LIN {X 0,Y 573.388,Z 194.884,A -85,B 0,C 180,E1 -2263.851,E2 -2263.851} C_VEL
LIN {X 0,Y 573.533,Z 175.271,A -85,B 0,C 180,E1 -2266.721,E2 -2266.721} C_VEL
LIN {X 0,Y 573.704,Z 157.685,A -85,B 0,C 180,E1 -2269.315,E2 -2269.315} C_VEL
LIN {X 0,Y 573.895,Z 140.113,A -85,B 0,C 180,E1 -2271.932,E2 -2271.932} C_VEL
LIN {X 0,Y 573.247,Z 134.603,A -85,B 0,C 180,E1 -2272.789,E2 -2272.789} C_VEL
LIN {X 0,Y 573.229,Z 134.582,A -85,B 0,C 180,E1 -2275.411,E2 -2275.411} C_VEL
LIN {X 0,Y 573.202,Z 134.579,A -85,B 0,C 180,E1 -2278.019,E2 -2278.019} C_VEL
LIN {X 0,Y 573.22,Z 134.577,A -85,B 0,C 180,E1 -2280.178,E2 -2280.178} C_VEL
LIN {X 0,Y 573.246,Z 134.579,A -85,B 0,C 180,E1 -2282.645,E2 -2282.645} C_VEL
LIN {X 0,Y 573.203,Z 134.583,A -85,B 0,C 180,E1 -2285.188,E2 -2285.188} C_VEL
LIN {X 0,Y 573.23,Z 134.575,A -85,B 0,C 180,E1 -2287.808,E2 -2287.808} C_VEL
LIN {X 0,Y 573.245,Z 134.58,A -85,B 0,C 180,E1 -2290.525,E2 -2290.525} C_VEL
LIN {X 0,Y 573.208,Z 134.579,A -85,B 0,C 180,E1 -2293.362,E2 -2293.362} C_VEL
LIN {X 0,Y 573.235,Z 134.581,A -85,B 0,C 180,E1 -2296.332,E2 -2296.332} C_VEL
LIN {X 0,Y 573.245,Z 134.574,A -85,B 0,C 180,E1 -2299.475,E2 -2299.475} C_VEL
LIN {X 0,Y 573.229,Z 134.583,A -85,B 0,C 180,E1 -2302.192,E2 -2302.192} C_VEL
LIN {X 0,Y 573.232,Z 134.575,A -85,B 0,C 180,E1 -2305.229,E2 -2305.229} C_VEL
LIN {X 0,Y 573.246,Z 134.577,A -85,B 0,C 180,E1 -2307.772,E2 -2307.772} C_VEL
LIN {X 0,Y 573.242,Z 134.576,A -85,B 0,C 180,E1 -2310.633,E2 -2310.633} C_VEL
LIN {X 0,Y 573.208,Z 134.578,A -85,B 0,C 180,E1 -2313.022,E2 -2313.022} C_VEL
LIN {X 0,Y 573.274,Z 134.572,A -85,B 0,C 180,E1 -2315.366,E2 -2315.366} C_VEL
LIN {X 0,Y 573.227,Z 134.578,A -85,B 0,C 180,E1 -2318.419,E2 -2318.419} C_VEL
LIN {X 0,Y 573.268,Z 134.571,A -85,B 0,C 180,E1 -2320.731,E2 -2320.731} C_VEL
LIN {X 0,Y 573.242,Z 134.582,A -85,B 0,C 180,E1 -2323.621,E2 -2323.621} C_VEL
LIN {X 0,Y 573.272,Z 134.578,A -85,B 0,C 180,E1 -2325.807,E2 -2325.807} C_VEL
LIN {X 0,Y 573.263,Z 134.572,A -85,B 0,C 180,E1 -2328.745,E2 -2328.745} C_VEL
LIN {X 0,Y 573.283,Z 134.578,A -85,B 0,C 180,E1 -2331.54,E2 -2331.54} C_VEL
LIN {X 0,Y 573.291,Z 134.568,A -85,B 0,C 180,E1 -2334.372,E2 -2334.372} C_VEL
LIN {X 0,Y 573.316,Z 134.566,A -85,B 0,C 180,E1 -2337.892,E2 -2337.892} C_VEL
LIN {X 0,Y 573.325,Z 134.566,A -85,B 0,C 180,E1 -2340.702,E2 -2340.702} C_VEL
LIN {X 0,Y 573.299,Z 134.571,A -85,B 0,C 180,E1 -2342.811,E2 -2342.811} C_VEL
LIN {X 0,Y 573.298,Z 134.569,A -85,B 0,C 180,E1 -2345.628,E2 -2345.628} C_VEL
LIN {X 0,Y 573.282,Z 134.571,A -85,B 0,C 180,E1 -2348.46,E2 -2348.46} C_VEL
LIN {X 0,Y 573.272,Z 134.574,A -85,B 0,C 180,E1 -2351.312,E2 -2351.312} C_VEL
LIN {X 0,Y 573.282,Z 134.573,A -85,B 0,C 180,E1 -2354.424,E2 -2354.424} C_VEL
LIN {X 0,Y 573.258,Z 134.576,A -85,B 0,C 180,E1 -2357.112,E2 -2357.112} C_VEL
LIN {X 0,Y 573.252,Z 134.575,A -85,B 0,C 180,E1 -2360.077,E2 -2360.077} C_VEL
LIN {X 0,Y 573.235,Z 134.577,A -85,B 0,C 180,E1 -2363.1,E2 -2363.1} C_VEL
LIN {X 0,Y 573.249,Z 134.577,A -85,B 0,C 180,E1 -2364.376,E2 -2364.376} C_VEL
LIN {X 0,Y 572.622,Z 134.659,A -85,B 0,C 180,E1 -2364.962,E2 -2364.962} C_VEL
LIN {X 0,Y 569.782,Z 135.012,A -85,B 0,C 180,E1 -2365.914,E2 -2365.914} C_VEL
LIN {X 0,Y 567.351,Z 135.314,A -85,B 0,C 180,E1 -2366.679,E2 -2366.679} C_VEL
LIN {X 0,Y 566.295,Z 135.44,A -85,B 0,C 180,E1 -2367.27,E2 -2367.27} C_VEL
LIN {X 0,Y 566.204,Z 135.451,A -85,B 0,C 180,E1 -2367.471,E2 -2367.471} C_VEL
LIN {X 0,Y 566.202,Z 135.453,A -85,B 0,C 180,E1 -2369.769,E2 -2369.769} C_VEL
LIN {X 0,Y 566.205,Z 135.458,A -85,B 0,C 180,E1 -2372.43,E2 -2372.43} C_VEL
LIN {X 0,Y 566.181,Z 135.454,A -85,B 0,C 180,E1 -2374.99,E2 -2374.99} C_VEL
LIN {X 0,Y 566.198,Z 135.453,A -85,B 0,C 180,E1 -2377.461,E2 -2377.461} C_VEL
LIN {X 0,Y 566.219,Z 135.456,A -85,B 0,C 180,E1 -2380.198,E2 -2380.198} C_VEL
LIN {X 0,Y 566.202,Z 135.451,A -85,B 0,C 180,E1 -2383.054,E2 -2383.054} C_VEL
LIN {X 0,Y 566.2,Z 135.458,A -85,B 0,C 180,E1 -2386.049,E2 -2386.049} C_VEL
LIN {X 0,Y 566.181,Z 135.454,A -85,B 0,C 180,E1 -2388.861,E2 -2388.861} C_VEL
LIN {X 0,Y 566.188,Z 135.462,A -85,B 0,C 180,E1 -2391.637,E2 -2391.637} C_VEL
LIN {X 0,Y 566.164,Z 135.457,A -85,B 0,C 180,E1 -2394.308,E2 -2394.308} C_VEL
LIN {X 0,Y 566.206,Z 135.452,A -85,B 0,C 180,E1 -2396.897,E2 -2396.897} C_VEL
LIN {X 0,Y 566.177,Z 135.463,A -85,B 0,C 180,E1 -2399.407,E2 -2399.407} C_VEL
LIN {X 0,Y 566.197,Z 135.454,A -85,B 0,C 180,E1 -2401.857,E2 -2401.857} C_VEL
LIN {X 0,Y 566.212,Z 135.451,A -85,B 0,C 180,E1 -2404.251,E2 -2404.251} C_VEL
LIN {X 0,Y 566.171,Z 135.458,A -85,B 0,C 180,E1 -2406.72,E2 -2406.72} C_VEL
LIN {X 0,Y 566.227,Z 135.456,A -85,B 0,C 180,E1 -2409.663,E2 -2409.663} C_VEL
LIN {X 0,Y 566.236,Z 135.473,A -85,B 0,C 180,E1 -2409.853,E2 -2409.853} C_VEL
LIN {X 0,Y 566.578,Z 139.18,A -85,B 0,C 180,E1 -2410.515,E2 -2410.515} C_VEL
LIN {X 0,Y 566.45,Z 154.128,A -85,B 0,C 180,E1 -2413.118,E2 -2413.118} C_VEL
LIN {X 0,Y 566.325,Z 171.323,A -85,B 0,C 180,E1 -2416.056,E2 -2416.056} C_VEL
LIN {X 0,Y 567.191,Z 177.354,A -85,B 0,C 180,E1 -2416.155,E2 -2416.155} C_VEL
LIN {X 0,Y 566.968,Z 277.969,A -85,B 0,C 180,E1 -2417.449,E2 -2417.449} C_VEL
LIN {X 0,Y 566.826,Z 291.223,A -85,B 0,C 180,E1 -2417.764,E2 -2417.764} C_VEL
LIN {X 0,Y 566.742,Z 303.381,A -85,B 0,C 180,E1 -2418.194,E2 -2418.194} C_VEL
LIN {X 0,Y 566.611,Z 315.58,A -85,B 0,C 180,E1 -2418.777,E2 -2418.777} C_VEL
LIN {X 0,Y 566.448,Z 326.553,A -85,B 0,C 180,E1 -2419.455,E2 -2419.455} C_VEL
LIN {X 0,Y 566.327,Z 337.072,A -85,B 0,C 180,E1 -2420.265,E2 -2420.265} C_VEL
LIN {X 0,Y 566.221,Z 345.669,A -85,B 0,C 180,E1 -2421.074,E2 -2421.074} C_VEL
LIN {X 0,Y 566.113,Z 353.59,A -85,B 0,C 180,E1 -2421.972,E2 -2421.972} C_VEL
LIN {X 0,Y 566.05,Z 360.158,A -85,B 0,C 180,E1 -2422.868,E2 -2422.868} C_VEL
LIN {X 0,Y 566.003,Z 366.627,A -85,B 0,C 180,E1 -2423.942,E2 -2423.942} C_VEL
LIN {X 0,Y 565.878,Z 371.764,A -85,B 0,C 180,E1 -2425.013,E2 -2425.013} C_VEL
LIN {X 0,Y 565.926,Z 375.754,A -85,B 0,C 180,E1 -2426.084,E2 -2426.084} C_VEL
LIN {X 0,Y 565.877,Z 378.703,A -85,B 0,C 180,E1 -2427.152,E2 -2427.152} C_VEL
LIN {X 0,Y 565.841,Z 380.126,A -85,B 0,C 180,E1 -2427.865,E2 -2427.865} C_VEL
LIN {X 0,Y 565.841,Z 381.757,A -85,B 0,C 180,E1 -2429.288,E2 -2429.288} C_VEL
LIN {X 0,Y 565.839,Z 381.996,A -85,B 0,C 180,E1 -2430,E2 -2430} C_VEL
LIN {X 0,Y 565.841,Z 381.815,A -85,B 0,C 180,E1 -2430.712,E2 -2430.712} C_VEL
LIN {X 0,Y 565.841,Z 380.266,A -85,B 0,C 180,E1 -2432.135,E2 -2432.135} C_VEL
LIN {X 0,Y 565.878,Z 378.906,A -85,B 0,C 180,E1 -2432.847,E2 -2432.847} C_VEL
LIN {X 0,Y 565.926,Z 376.029,A -85,B 0,C 180,E1 -2433.916,E2 -2433.916} C_VEL
LIN {X 0,Y 565.878,Z 372.129,A -85,B 0,C 180,E1 -2434.987,E2 -2434.987} C_VEL
LIN {X 0,Y 565.99,Z 367.097,A -85,B 0,C 180,E1 -2436.059,E2 -2436.059} C_VEL
LIN {X 0,Y 566.031,Z 360.772,A -85,B 0,C 180,E1 -2437.132,E2 -2437.132} C_VEL
LIN {X 0,Y 566.128,Z 352.85,A -85,B 0,C 180,E1 -2438.208,E2 -2438.208} C_VEL
LIN {X 0,Y 566.249,Z 342.998,A -85,B 0,C 180,E1 -2439.285,E2 -2439.285} C_VEL
LIN {X 0,Y 566.424,Z 332.68,A -85,B 0,C 180,E1 -2440.184,E2 -2440.184} C_VEL
LIN {X 0,Y 566.506,Z 321.342,A -85,B 0,C 180,E1 -2440.976,E2 -2440.976} C_VEL
LIN {X 0,Y 566.688,Z 310.188,A -85,B 0,C 180,E1 -2441.592,E2 -2441.592} C_VEL
LIN {X 0,Y 566.804,Z 297.595,A -85,B 0,C 180,E1 -2442.119,E2 -2442.119} C_VEL
LIN {X 0,Y 566.94,Z 284.42,A -85,B 0,C 180,E1 -2442.506,E2 -2442.506} C_VEL
LIN {X 0,Y 567.04,Z 272.054,A -85,B 0,C 180,E1 -2442.732,E2 -2442.732} C_VEL
LIN {X 0,Y 567.096,Z 176.029,A -85,B 0,C 180,E1 -2443.954,E2 -2443.954} C_VEL
LIN {X 0,Y 566.266,Z 171.009,A -85,B 0,C 180,E1 -2444.051,E2 -2444.051} C_VEL
LIN {X 0,Y 566.442,Z 154.652,A -85,B 0,C 180,E1 -2446.883,E2 -2446.883} C_VEL
LIN {X 0,Y 566.561,Z 139.725,A -85,B 0,C 180,E1 -2449.48,E2 -2449.48} C_VEL
LIN {X 0,Y 566.215,Z 135.457,A -85,B 0,C 180,E1 -2450.242,E2 -2450.242} C_VEL
LIN {X 0,Y 566.175,Z 135.462,A -85,B 0,C 180,E1 -2452.632,E2 -2452.632} C_VEL
LIN {X 0,Y 566.221,Z 135.455,A -85,B 0,C 180,E1 -2455.03,E2 -2455.03} C_VEL
LIN {X 0,Y 566.209,Z 135.452,A -85,B 0,C 180,E1 -2457.339,E2 -2457.339} C_VEL
LIN {X 0,Y 566.199,Z 135.451,A -85,B 0,C 180,E1 -2459.769,E2 -2459.769} C_VEL
LIN {X 0,Y 566.204,Z 135.458,A -85,B 0,C 180,E1 -2462.429,E2 -2462.429} C_VEL
LIN {X 0,Y 566.181,Z 135.456,A -85,B 0,C 180,E1 -2464.989,E2 -2464.989} C_VEL
LIN {X 0,Y 566.197,Z 135.452,A -85,B 0,C 180,E1 -2467.461,E2 -2467.461} C_VEL
LIN {X 0,Y 566.208,Z 135.458,A -85,B 0,C 180,E1 -2470.199,E2 -2470.199} C_VEL
LIN {X 0,Y 566.203,Z 135.451,A -85,B 0,C 180,E1 -2473.054,E2 -2473.054} C_VEL
LIN {X 0,Y 566.199,Z 135.459,A -85,B 0,C 180,E1 -2476.048,E2 -2476.048} C_VEL
LIN {X 0,Y 566.221,Z 135.449,A -85,B 0,C 180,E1 -2479.212,E2 -2479.212} C_VEL
LIN {X 0,Y 566.19,Z 135.457,A -85,B 0,C 180,E1 -2481.637,E2 -2481.637} C_VEL
LIN {X 0,Y 566.162,Z 135.46,A -85,B 0,C 180,E1 -2484.308,E2 -2484.308} C_VEL
LIN {X 0,Y 566.22,Z 135.449,A -85,B 0,C 180,E1 -2486.898,E2 -2486.898} C_VEL
LIN {X 0,Y 566.181,Z 135.458,A -85,B 0,C 180,E1 -2489.407,E2 -2489.407} C_VEL
LIN {X 0,Y 566.211,Z 135.457,A -85,B 0,C 180,E1 -2491.857,E2 -2491.857} C_VEL
LIN {X 0,Y 566.214,Z 135.451,A -85,B 0,C 180,E1 -2494.251,E2 -2494.251} C_VEL
LIN {X 0,Y 566.172,Z 135.455,A -85,B 0,C 180,E1 -2496.718,E2 -2496.718} C_VEL
LIN {X 0,Y 566.214,Z 135.456,A -85,B 0,C 180,E1 -2499.663,E2 -2499.663} C_VEL
LIN {X 0,Y 566.199,Z 135.452,A -85,B 0,C 180,E1 -2502.668,E2 -2502.668} C_VEL
LIN {X 0,Y 566.234,Z 135.451,A -85,B 0,C 180,E1 -2505.627,E2 -2505.627} C_VEL
LIN {X 0,Y 566.234,Z 135.45,A -85,B 0,C 180,E1 -2508.675,E2 -2508.675} C_VEL
LIN {X 0,Y 566.226,Z 135.452,A -85,B 0,C 180,E1 -2511.434,E2 -2511.434} C_VEL
LIN {X 0,Y 566.264,Z 135.444,A -85,B 0,C 180,E1 -2514.302,E2 -2514.302} C_VEL
LIN {X 0,Y 566.284,Z 135.441,A -85,B 0,C 180,E1 -2517.866,E2 -2517.866} C_VEL
LIN {X 0,Y 566.305,Z 135.447,A -85,B 0,C 180,E1 -2520.711,E2 -2520.711} C_VEL
LIN {X 0,Y 566.271,Z 135.45,A -85,B 0,C 180,E1 -2522.846,E2 -2522.846} C_VEL
LIN {X 0,Y 566.261,Z 135.444,A -85,B 0,C 180,E1 -2525.698,E2 -2525.698} C_VEL
LIN {X 0,Y 566.227,Z 135.458,A -85,B 0,C 180,E1 -2528.566,E2 -2528.566} C_VEL
LIN {X 0,Y 566.241,Z 135.446,A -85,B 0,C 180,E1 -2531.454,E2 -2531.454} C_VEL
LIN {X 0,Y 566.233,Z 135.455,A -85,B 0,C 180,E1 -2534.507,E2 -2534.507} C_VEL
LIN {X 0,Y 566.197,Z 135.452,A -85,B 0,C 180,E1 -2537.332,E2 -2537.332} C_VEL
LIN {X 0,Y 566.205,Z 135.458,A -85,B 0,C 180,E1 -2540.338,E2 -2540.338} C_VEL
LIN {X 0,Y 566.168,Z 135.455,A -85,B 0,C 180,E1 -2543.281,E2 -2543.281} C_VEL
LIN {X 0,Y 566.206,Z 135.456,A -85,B 0,C 180,E1 -2545.749,E2 -2545.749} C_VEL
LIN {X 0,Y 566.202,Z 135.457,A -85,B 0,C 180,E1 -2548.202,E2 -2548.202} C_VEL
LIN {X 0,Y 566.187,Z 135.453,A -85,B 0,C 180,E1 -2551.076,E2 -2551.076} C_VEL
LIN {X 0,Y 566.211,Z 135.459,A -85,B 0,C 180,E1 -2553.734,E2 -2553.734} C_VEL
LIN {X 0,Y 566.181,Z 135.454,A -85,B 0,C 180,E1 -2556.571,E2 -2556.571} C_VEL
LIN {X 0,Y 566.216,Z 135.458,A -85,B 0,C 180,E1 -2559.686,E2 -2559.686} C_VEL
LIN {X 0,Y 566.192,Z 135.454,A -85,B 0,C 180,E1 -2562.916,E2 -2562.916} C_VEL
LIN {X 0,Y 566.159,Z 135.458,A -85,B 0,C 180,E1 -2565.961,E2 -2565.961} C_VEL
LIN {X 0,Y 566.178,Z 135.454,A -85,B 0,C 180,E1 -2568.141,E2 -2568.141} C_VEL
LIN {X 0,Y 566.209,Z 135.452,A -85,B 0,C 180,E1 -2570.726,E2 -2570.726} C_VEL
LIN {X 0,Y 566.183,Z 135.455,A -85,B 0,C 180,E1 -2573.789,E2 -2573.789} C_VEL
LIN {X 0,Y 566.197,Z 135.452,A -85,B 0,C 180,E1 -2576.269,E2 -2576.269} C_VEL
LIN {X 0,Y 566.182,Z 135.462,A -85,B 0,C 180,E1 -2578.926,E2 -2578.926} C_VEL
LIN {X 0,Y 566.152,Z 135.458,A -85,B 0,C 180,E1 -2581.854,E2 -2581.854} C_VEL
LIN {X 0,Y 566.19,Z 135.456,A -85,B 0,C 180,E1 -2584.25,E2 -2584.25} C_VEL
LIN {X 0,Y 566.22,Z 135.65,A -85,B 0,C 180,E1 -2587.097,E2 -2587.097} C_VEL
LIN {X 0,Y 566.926,Z 139.96,A -85,B 0,C 180,E1 -2587.784,E2 -2587.784} C_VEL
LIN {X 0,Y 566.724,Z 157.527,A -85,B 0,C 180,E1 -2590.438,E2 -2590.438} C_VEL
LIN {X 0,Y 566.533,Z 175.433,A -85,B 0,C 180,E1 -2593.103,E2 -2593.103} C_VEL
LIN {X 0,Y 566.396,Z 195.149,A -85,B 0,C 180,E1 -2595.998,E2 -2595.998} C_VEL
LIN {X 0,Y 567.166,Z 202.303,A -85,B 0,C 180,E1 -2596.109,E2 -2596.109} C_VEL
LIN {X 0,Y 566.943,Z 302.95,A -85,B 0,C 180,E1 -2597.403,E2 -2597.403} C_VEL
LIN {X 0,Y 566.836,Z 316.22,A -85,B 0,C 180,E1 -2597.719,E2 -2597.719} C_VEL
LIN {X 0,Y 566.729,Z 328.379,A -85,B 0,C 180,E1 -2598.148,E2 -2598.148} C_VEL
LIN {X 0,Y 566.589,Z 340.453,A -85,B 0,C 180,E1 -2598.724,E2 -2598.724} C_VEL
LIN {X 0,Y 566.439,Z 352.197,A -85,B 0,C 180,E1 -2599.455,E2 -2599.455} C_VEL
LIN {X 0,Y 566.325,Z 362.605,A -85,B 0,C 180,E1 -2600.266,E2 -2600.266} C_VEL
LIN {X 0,Y 566.207,Z 371.114,A -85,B 0,C 180,E1 -2601.074,E2 -2601.074} C_VEL
LIN {X 0,Y 566.112,Z 378.961,A -85,B 0,C 180,E1 -2601.972,E2 -2601.972} C_VEL
LIN {X 0,Y 566.003,Z 386.623,A -85,B 0,C 180,E1 -2603.047,E2 -2603.047} C_VEL
LIN {X 0,Y 566.004,Z 393.68,A -85,B 0,C 180,E1 -2604.299,E2 -2604.299} C_VEL
LIN {X 0,Y 565.933,Z 398.373,A -85,B 0,C 180,E1 -2605.37,E2 -2605.37} C_VEL
LIN {X 0,Y 565.927,Z 401.958,A -85,B 0,C 180,E1 -2606.44,E2 -2606.44} C_VEL
LIN {X 0,Y 565.878,Z 403.808,A -85,B 0,C 180,E1 -2607.152,E2 -2607.152} C_VEL
LIN {X 0,Y 565.846,Z 406.184,A -85,B 0,C 180,E1 -2608.577,E2 -2608.577} C_VEL
LIN {X 0,Y 565.839,Z 407,A -85,B 0,C 180,E1 -2610,E2 -2610} C_VEL
LIN {X 0,Y 565.846,Z 406.185,A -85,B 0,C 180,E1 -2611.423,E2 -2611.423} C_VEL
LIN {X 0,Y 565.878,Z 403.81,A -85,B 0,C 180,E1 -2612.848,E2 -2612.848} C_VEL
LIN {X 0,Y 565.926,Z 400.895,A -85,B 0,C 180,E1 -2613.916,E2 -2613.916} C_VEL
LIN {X 0,Y 565.878,Z 396.948,A -85,B 0,C 180,E1 -2614.987,E2 -2614.987} C_VEL
LIN {X 0,Y 566.002,Z 391.867,A -85,B 0,C 180,E1 -2616.059,E2 -2616.059} C_VEL
LIN {X 0,Y 566.04,Z 385.467,A -85,B 0,C 180,E1 -2617.132,E2 -2617.132} C_VEL
LIN {X 0,Y 566.134,Z 377.477,A -85,B 0,C 180,E1 -2618.208,E2 -2618.208} C_VEL
LIN {X 0,Y 566.229,Z 369.334,A -85,B 0,C 180,E1 -2619.105,E2 -2619.105} C_VEL
LIN {X 0,Y 566.347,Z 359.398,A -85,B 0,C 180,E1 -2620.005,E2 -2620.005} C_VEL
LIN {X 0,Y 566.536,Z 348.291,A -85,B 0,C 180,E1 -2620.807,E2 -2620.807} C_VEL
LIN {X 0,Y 566.613,Z 337.173,A -85,B 0,C 180,E1 -2621.447,E2 -2621.447} C_VEL
LIN {X 0,Y 566.745,Z 324.979,A -85,B 0,C 180,E1 -2621.988,E2 -2621.988} C_VEL
LIN {X 0,Y 566.887,Z 312.174,A -85,B 0,C 180,E1 -2622.394,E2 -2622.394} C_VEL
LIN {X 0,Y 567.016,Z 298.601,A -85,B 0,C 180,E1 -2622.664,E2 -2622.664} C_VEL
LIN {X 0,Y 567.043,Z 199.392,A -85,B 0,C 180,E1 -2623.932,E2 -2623.932} C_VEL
LIN {X 0,Y 566.384,Z 194.884,A -85,B 0,C 180,E1 -2624.026,E2 -2624.026} C_VEL
LIN {X 0,Y 566.547,Z 174.047,A -85,B 0,C 180,E1 -2627.102,E2 -2627.102} C_VEL
LIN {X 0,Y 566.776,Z 155.018,A -85,B 0,C 180,E1 -2629.938,E2 -2629.938} C_VEL
LIN {X 0,Y 566.926,Z 139.958,A -85,B 0,C 180,E1 -2632.216,E2 -2632.216} C_VEL
LIN {X 0,Y 566.202,Z 135.46,A -85,B 0,C 180,E1 -2632.95,E2 -2632.95} C_VEL
LIN {X 0,Y 566.191,Z 135.455,A -85,B 0,C 180,E1 -2635.75,E2 -2635.75} C_VEL
LIN {X 0,Y 566.151,Z 135.457,A -85,B 0,C 180,E1 -2638.192,E2 -2638.192} C_VEL
LIN {X 0,Y 566.182,Z 135.462,A -85,B 0,C 180,E1 -2641.074,E2 -2641.074} C_VEL
LIN {X 0,Y 566.197,Z 135.452,A -85,B 0,C 180,E1 -2643.731,E2 -2643.731} C_VEL
LIN {X 0,Y 566.199,Z 135.457,A -85,B 0,C 180,E1 -2646.57,E2 -2646.57} C_VEL
LIN {X 0,Y 566.209,Z 135.45,A -85,B 0,C 180,E1 -2649.685,E2 -2649.685} C_VEL
LIN {X 0,Y 566.184,Z 135.455,A -85,B 0,C 180,E1 -2652.09,E2 -2652.09} C_VEL
LIN {X 0,Y 566.164,Z 135.459,A -85,B 0,C 180,E1 -2655.037,E2 -2655.037} C_VEL
LIN {X 0,Y 566.176,Z 135.456,A -85,B 0,C 180,E1 -2657.909,E2 -2657.909} C_VEL
LIN {X 0,Y 566.216,Z 135.454,A -85,B 0,C 180,E1 -2660.726,E2 -2660.726} C_VEL
LIN {X 0,Y 566.182,Z 135.454,A -85,B 0,C 180,E1 -2663.429,E2 -2663.429} C_VEL
LIN {X 0,Y 566.211,Z 135.459,A -85,B 0,C 180,E1 -2666.266,E2 -2666.266} C_VEL
LIN {X 0,Y 566.185,Z 135.454,A -85,B 0,C 180,E1 -2668.924,E2 -2668.924} C_VEL
LIN {X 0,Y 566.19,Z 135.459,A -85,B 0,C 180,E1 -2671.856,E2 -2671.856} C_VEL
LIN {X 0,Y 566.237,Z 135.447,A -85,B 0,C 180,E1 -2675.039,E2 -2675.039} C_VEL
LIN {X 0,Y 566.192,Z 135.458,A -85,B 0,C 180,E1 -2678.137,E2 -2678.137} C_VEL
LIN {X 0,Y 566.23,Z 135.448,A -85,B 0,C 180,E1 -2680.614,E2 -2680.614} C_VEL
LIN {X 0,Y 566.209,Z 135.455,A -85,B 0,C 180,E1 -2683.412,E2 -2683.412} C_VEL
LIN {X 0,Y 566.193,Z 135.453,A -85,B 0,C 180,E1 -2686.359,E2 -2686.359} C_VEL
LIN {X 0,Y 566.235,Z 135.447,A -85,B 0,C 180,E1 -2688.675,E2 -2688.675} C_VEL
LIN {X 0,Y 566.227,Z 135.457,A -85,B 0,C 180,E1 -2691.434,E2 -2691.434} C_VEL
LIN {X 0,Y 566.261,Z 135.444,A -85,B 0,C 180,E1 -2694.302,E2 -2694.302} C_VEL
LIN {X 0,Y 566.286,Z 135.442,A -85,B 0,C 180,E1 -2697.866,E2 -2697.866} C_VEL
LIN {X 0,Y 566.296,Z 135.442,A -85,B 0,C 180,E1 -2700.711,E2 -2700.711} C_VEL
LIN {X 0,Y 566.267,Z 135.448,A -85,B 0,C 180,E1 -2702.846,E2 -2702.846} C_VEL
LIN {X 0,Y 566.264,Z 135.444,A -85,B 0,C 180,E1 -2705.698,E2 -2705.698} C_VEL
LIN {X 0,Y 566.226,Z 135.451,A -85,B 0,C 180,E1 -2708.566,E2 -2708.566} C_VEL
LIN {X 0,Y 566.242,Z 135.448,A -85,B 0,C 180,E1 -2711.454,E2 -2711.454} C_VEL
LIN {X 0,Y 566.234,Z 135.452,A -85,B 0,C 180,E1 -2714.507,E2 -2714.507} C_VEL
LIN {X 0,Y 566.199,Z 135.453,A -85,B 0,C 180,E1 -2717.332,E2 -2717.332} C_VEL
LIN {X 0,Y 566.214,Z 135.455,A -85,B 0,C 180,E1 -2720.337,E2 -2720.337} C_VEL
LIN {X 0,Y 566.173,Z 135.455,A -85,B 0,C 180,E1 -2723.282,E2 -2723.282} C_VEL
LIN {X 0,Y 566.214,Z 135.45,A -85,B 0,C 180,E1 -2725.749,E2 -2725.749} C_VEL
LIN {X 0,Y 566.204,Z 135.451,A -85,B 0,C 180,E1 -2727.471,E2 -2727.471} C_VEL
LIN {X 0,Y 565.523,Z 135.542,A -85,B 0,C 180,E1 -2728.064,E2 -2728.064} C_VEL
LIN {X 0,Y 562.658,Z 135.898,A -85,B 0,C 180,E1 -2729.028,E2 -2729.028} C_VEL
LIN {X 0,Y 560.248,Z 136.198,A -85,B 0,C 180,E1 -2729.804,E2 -2729.804} C_VEL
LIN {X 0,Y 559.22,Z 136.329,A -85,B 0,C 180,E1 -2730.402,E2 -2730.402} C_VEL
LIN {X 0,Y 559.14,Z 136.333,A -85,B 0,C 180,E1 -2730.605,E2 -2730.605} C_VEL
LIN {X 0,Y 559.158,Z 136.331,A -85,B 0,C 180,E1 -2732.715,E2 -2732.715} C_VEL
LIN {X 0,Y 559.128,Z 136.332,A -85,B 0,C 180,E1 -2735.324,E2 -2735.324} C_VEL
LIN {X 0,Y 559.136,Z 136.34,A -85,B 0,C 180,E1 -2738.018,E2 -2738.018} C_VEL
LIN {X 0,Y 559.176,Z 136.327,A -85,B 0,C 180,E1 -2740.811,E2 -2740.811} C_VEL
LIN {X 0,Y 559.143,Z 136.337,A -85,B 0,C 180,E1 -2743.734,E2 -2743.734} C_VEL
LIN {X 0,Y 559.148,Z 136.33,A -85,B 0,C 180,E1 -2746.804,E2 -2746.804} C_VEL
LIN {X 0,Y 559.159,Z 136.33,A -85,B 0,C 180,E1 -2749.188,E2 -2749.188} C_VEL
LIN {X 0,Y 559.135,Z 136.336,A -85,B 0,C 180,E1 -2751.983,E2 -2751.983} C_VEL
LIN {X 0,Y 559.133,Z 136.332,A -85,B 0,C 180,E1 -2754.788,E2 -2754.788} C_VEL
LIN {X 0,Y 559.156,Z 136.336,A -85,B 0,C 180,E1 -2757.365,E2 -2757.365} C_VEL
LIN {X 0,Y 559.147,Z 136.331,A -85,B 0,C 180,E1 -2760.144,E2 -2760.144} C_VEL
LIN {X 0,Y 559.171,Z 136.332,A -85,B 0,C 180,E1 -2763.098,E2 -2763.098} C_VEL
LIN {X 0,Y 559.157,Z 136.336,A -85,B 0,C 180,E1 -2765.495,E2 -2765.495} C_VEL
LIN {X 0,Y 559.175,Z 136.33,A -85,B 0,C 180,E1 -2768.624,E2 -2768.624} C_VEL
LIN {X 0,Y 559.206,Z 136.54,A -85,B 0,C 180,E1 -2769.781,E2 -2769.781} C_VEL
LIN {X 0,Y 559.602,Z 139.823,A -85,B 0,C 180,E1 -2770.377,E2 -2770.377} C_VEL
LIN {X 0,Y 559.445,Z 154.46,A -85,B 0,C 180,E1 -2772.952,E2 -2772.952} C_VEL
LIN {X 0,Y 559.265,Z 171.126,A -85,B 0,C 180,E1 -2775.862,E2 -2775.862} C_VEL
LIN {X 0,Y 560.28,Z 177.505,A -85,B 0,C 180,E1 -2775.981,E2 -2775.981} C_VEL
LIN {X 0,Y 560.042,Z 278.042,A -85,B 0,C 180,E1 -2777.291,E2 -2777.291} C_VEL
LIN {X 0,Y 559.91,Z 291.273,A -85,B 0,C 180,E1 -2777.61,E2 -2777.61} C_VEL
LIN {X 0,Y 559.787,Z 303.408,A -85,B 0,C 180,E1 -2778.045,E2 -2778.045} C_VEL
LIN {X 0,Y 559.649,Z 315.083,A -85,B 0,C 180,E1 -2778.607,E2 -2778.607} C_VEL
LIN {X 0,Y 559.474,Z 326.559,A -85,B 0,C 180,E1 -2779.322,E2 -2779.322} C_VEL
LIN {X 0,Y 559.308,Z 337.077,A -85,B 0,C 180,E1 -2780.142,E2 -2780.142} C_VEL
LIN {X 0,Y 559.197,Z 345.674,A -85,B 0,C 180,E1 -2780.961,E2 -2780.961} C_VEL
LIN {X 0,Y 559.05,Z 353.595,A -85,B 0,C 180,E1 -2781.87,E2 -2781.87} C_VEL
LIN {X 0,Y 558.971,Z 361.457,A -85,B 0,C 180,E1 -2782.977,E2 -2782.977} C_VEL
LIN {X 0,Y 558.936,Z 368.454,A -85,B 0,C 180,E1 -2784.227,E2 -2784.227} C_VEL
LIN {X 0,Y 558.826,Z 373.195,A -85,B 0,C 180,E1 -2785.311,E2 -2785.311} C_VEL
LIN {X 0,Y 558.836,Z 376.828,A -85,B 0,C 180,E1 -2786.395,E2 -2786.395} C_VEL
LIN {X 0,Y 558.799,Z 378.705,A -85,B 0,C 180,E1 -2787.116,E2 -2787.116} C_VEL
LIN {X 0,Y 558.747,Z 380.126,A -85,B 0,C 180,E1 -2787.837,E2 -2787.837} C_VEL
LIN {X 0,Y 558.741,Z 381.756,A -85,B 0,C 180,E1 -2789.279,E2 -2789.279} C_VEL
LIN {X 0,Y 558.74,Z 381.996,A -85,B 0,C 180,E1 -2790,E2 -2790} C_VEL
LIN {X 0,Y 558.741,Z 381.815,A -85,B 0,C 180,E1 -2790.721,E2 -2790.721} C_VEL
LIN {X 0,Y 558.747,Z 380.264,A -85,B 0,C 180,E1 -2792.162,E2 -2792.162} C_VEL
LIN {X 0,Y 558.8,Z 378.904,A -85,B 0,C 180,E1 -2792.884,E2 -2792.884} C_VEL
LIN {X 0,Y 558.844,Z 376.027,A -85,B 0,C 180,E1 -2793.966,E2 -2793.966} C_VEL
LIN {X 0,Y 558.798,Z 372.127,A -85,B 0,C 180,E1 -2795.051,E2 -2795.051} C_VEL
LIN {X 0,Y 558.91,Z 367.095,A -85,B 0,C 180,E1 -2796.136,E2 -2796.136} C_VEL
LIN {X 0,Y 558.972,Z 360.768,A -85,B 0,C 180,E1 -2797.223,E2 -2797.223} C_VEL
LIN {X 0,Y 559.091,Z 352.845,A -85,B 0,C 180,E1 -2798.312,E2 -2798.312} C_VEL
LIN {X 0,Y 559.224,Z 342.992,A -85,B 0,C 180,E1 -2799.403,E2 -2799.403} C_VEL
LIN {X 0,Y 559.429,Z 332.67,A -85,B 0,C 180,E1 -2800.313,E2 -2800.313} C_VEL
LIN {X 0,Y 559.535,Z 321.62,A -85,B 0,C 180,E1 -2801.096,E2 -2801.096} C_VEL
LIN {X 0,Y 559.726,Z 310.178,A -85,B 0,C 180,E1 -2801.738,E2 -2801.738} C_VEL
LIN {X 0,Y 559.881,Z 297.601,A -85,B 0,C 180,E1 -2802.271,E2 -2802.271} C_VEL
LIN {X 0,Y 560.009,Z 284.435,A -85,B 0,C 180,E1 -2802.664,E2 -2802.664} C_VEL
LIN {X 0,Y 560.131,Z 272.058,A -85,B 0,C 180,E1 -2802.891,E2 -2802.891} C_VEL
LIN {X 0,Y 560.211,Z 176.66,A -85,B 0,C 180,E1 -2804.122,E2 -2804.122} C_VEL
LIN {X 0,Y 559.247,Z 171.101,A -85,B 0,C 180,E1 -2804.231,E2 -2804.231} C_VEL
LIN {X 0,Y 559.445,Z 154.987,A -85,B 0,C 180,E1 -2807.048,E2 -2807.048} C_VEL
LIN {X 0,Y 559.592,Z 140.346,A -85,B 0,C 180,E1 -2809.62,E2 -2809.62} C_VEL
LIN {X 0,Y 559.17,Z 136.335,A -85,B 0,C 180,E1 -2810.365,E2 -2810.365} C_VEL
LIN {X 0,Y 559.138,Z 136.334,A -85,B 0,C 180,E1 -2813.427,E2 -2813.427} C_VEL
LIN {X 0,Y 559.18,Z 136.328,A -85,B 0,C 180,E1 -2816.097,E2 -2816.097} C_VEL
LIN {X 0,Y 559.164,Z 136.335,A -85,B 0,C 180,E1 -2818.529,E2 -2818.529} C_VEL
LIN {X 0,Y 559.145,Z 136.331,A -85,B 0,C 180,E1 -2821.272,E2 -2821.272} C_VEL
LIN {X 0,Y 559.158,Z 136.33,A -85,B 0,C 180,E1 -2823.947,E2 -2823.947} C_VEL
LIN {X 0,Y 559.142,Z 136.331,A -85,B 0,C 180,E1 -2827.108,E2 -2827.108} C_VEL
LIN {X 0,Y 559.162,Z 136.332,A -85,B 0,C 180,E1 -2829.941,E2 -2829.941} C_VEL
LIN {X 0,Y 559.162,Z 136.331,A -85,B 0,C 180,E1 -2832.743,E2 -2832.743} C_VEL
LIN {X 0,Y 559.154,Z 136.333,A -85,B 0,C 180,E1 -2835.76,E2 -2835.76} C_VEL
LIN {X 0,Y 559.166,Z 136.335,A -85,B 0,C 180,E1 -2838.23,E2 -2838.23} C_VEL
LIN {X 0,Y 559.179,Z 136.326,A -85,B 0,C 180,E1 -2841.191,E2 -2841.191} C_VEL
LIN {X 0,Y 559.139,Z 136.338,A -85,B 0,C 180,E1 -2843.789,E2 -2843.789} C_VEL
LIN {X 0,Y 559.163,Z 136.33,A -85,B 0,C 180,E1 -2846.425,E2 -2846.425} C_VEL
LIN {X 0,Y 559.155,Z 136.329,A -85,B 0,C 180,E1 -2848.98,E2 -2848.98} C_VEL
LIN {X 0,Y 559.168,Z 136.336,A -85,B 0,C 180,E1 -2851.619,E2 -2851.619} C_VEL
LIN {X 0,Y 559.181,Z 136.331,A -85,B 0,C 180,E1 -2853.903,E2 -2853.903} C_VEL
LIN {X 0,Y 559.142,Z 136.33,A -85,B 0,C 180,E1 -2856.571,E2 -2856.571} C_VEL
LIN {X 0,Y 559.18,Z 136.335,A -85,B 0,C 180,E1 -2859.395,E2 -2859.395} C_VEL
LIN {X 0,Y 559.147,Z 136.335,A -85,B 0,C 180,E1 -2861.686,E2 -2861.686} C_VEL
LIN {X 0,Y 559.165,Z 136.329,A -85,B 0,C 180,E1 -2863.948,E2 -2863.948} C_VEL
LIN {X 0,Y 559.171,Z 136.327,A -85,B 0,C 180,E1 -2866.184,E2 -2866.184} C_VEL
LIN {X 0,Y 559.195,Z 136.334,A -85,B 0,C 180,E1 -2869.133,E2 -2869.133} C_VEL
LIN {X 0,Y 559.203,Z 136.323,A -85,B 0,C 180,E1 -2872.054,E2 -2872.054} C_VEL
LIN {X 0,Y 559.251,Z 136.327,A -85,B 0,C 180,E1 -2874.953,E2 -2874.953} C_VEL
LIN {X 0,Y 559.255,Z 136.316,A -85,B 0,C 180,E1 -2877.839,E2 -2877.839} C_VEL
LIN {X 0,Y 559.275,Z 136.323,A -85,B 0,C 180,E1 -2880.72,E2 -2880.72} C_VEL
LIN {X 0,Y 559.237,Z 136.326,A -85,B 0,C 180,E1 -2882.881,E2 -2882.881} C_VEL
LIN {X 0,Y 559.23,Z 136.32,A -85,B 0,C 180,E1 -2885.77,E2 -2885.77} C_VEL
LIN {X 0,Y 559.186,Z 136.333,A -85,B 0,C 180,E1 -2888.674,E2 -2888.674} C_VEL
LIN {X 0,Y 559.204,Z 136.323,A -85,B 0,C 180,E1 -2891.6,E2 -2891.6} C_VEL
LIN {X 0,Y 559.199,Z 136.329,A -85,B 0,C 180,E1 -2894.596,E2 -2894.596} C_VEL
LIN {X 0,Y 559.14,Z 136.331,A -85,B 0,C 180,E1 -2897.558,E2 -2897.558} C_VEL
LIN {X 0,Y 559.164,Z 136.332,A -85,B 0,C 180,E1 -2899.838,E2 -2899.838} C_VEL
LIN {X 0,Y 559.14,Z 136.34,A -85,B 0,C 180,E1 -2902.153,E2 -2902.153} C_VEL
LIN {X 0,Y 559.174,Z 136.327,A -85,B 0,C 180,E1 -2905.298,E2 -2905.298} C_VEL
LIN {X 0,Y 559.137,Z 136.337,A -85,B 0,C 180,E1 -2907.715,E2 -2907.715} C_VEL
LIN {X 0,Y 559.15,Z 136.334,A -85,B 0,C 180,E1 -2910.183,E2 -2910.183} C_VEL
LIN {X 0,Y 559.155,Z 136.329,A -85,B 0,C 180,E1 -2912.715,E2 -2912.715} C_VEL
LIN {X 0,Y 559.122,Z 136.336,A -85,B 0,C 180,E1 -2915.325,E2 -2915.325} C_VEL
LIN {X 0,Y 559.129,Z 136.336,A -85,B 0,C 180,E1 -2918.018,E2 -2918.018} C_VEL
LIN {X 0,Y 559.154,Z 136.33,A -85,B 0,C 180,E1 -2920.813,E2 -2920.813} C_VEL
LIN {X 0,Y 559.135,Z 136.337,A -85,B 0,C 180,E1 -2923.735,E2 -2923.735} C_VEL
LIN {X 0,Y 559.131,Z 136.334,A -85,B 0,C 180,E1 -2926.805,E2 -2926.805} C_VEL
LIN {X 0,Y 559.153,Z 136.337,A -85,B 0,C 180,E1 -2929.188,E2 -2929.188} C_VEL
LIN {X 0,Y 559.129,Z 136.333,A -85,B 0,C 180,E1 -2931.982,E2 -2931.982} C_VEL
LIN {X 0,Y 559.13,Z 136.336,A -85,B 0,C 180,E1 -2934.788,E2 -2934.788} C_VEL
LIN {X 0,Y 559.149,Z 136.335,A -85,B 0,C 180,E1 -2937.366,E2 -2937.366} C_VEL
LIN {X 0,Y 559.112,Z 136.336,A -85,B 0,C 180,E1 -2940.15,E2 -2940.15} C_VEL
LIN {X 0,Y 559.142,Z 136.337,A -85,B 0,C 180,E1 -2943.179,E2 -2943.179} C_VEL
LIN {X 0,Y 559.115,Z 136.338,A -85,B 0,C 180,E1 -2945.493,E2 -2945.493} C_VEL
LIN {X 0,Y 559.16,Z 136.353,A -85,B 0,C 180,E1 -2946.924,E2 -2946.924} C_VEL
LIN {X 0,Y 560.003,Z 142.318,A -85,B 0,C 180,E1 -2947.883,E2 -2947.883} C_VEL
LIN {X 0,Y 559.758,Z 159.109,A -85,B 0,C 180,E1 -2950.449,E2 -2950.449} C_VEL
LIN {X 0,Y 559.514,Z 177.43,A -85,B 0,C 180,E1 -2953.208,E2 -2953.208} C_VEL
LIN {X 0,Y 559.387,Z 195.058,A -85,B 0,C 180,E1 -2955.819,E2 -2955.819} C_VEL
LIN {X 0,Y 560.27,Z 202.239,A -85,B 0,C 180,E1 -2955.934,E2 -2955.934} C_VEL
LIN {X 0,Y 560.03,Z 302.948,A -85,B 0,C 180,E1 -2957.245,E2 -2957.245} C_VEL
LIN {X 0,Y 559.894,Z 316.219,A -85,B 0,C 180,E1 -2957.564,E2 -2957.564} C_VEL
LIN {X 0,Y 559.78,Z 329.499,A -85,B 0,C 180,E1 -2958.045,E2 -2958.045} C_VEL
LIN {X 0,Y 559.601,Z 341.44,A -85,B 0,C 180,E1 -2958.639,E2 -2958.639} C_VEL
LIN {X 0,Y 559.426,Z 353.485,A -85,B 0,C 180,E1 -2959.413,E2 -2959.413} C_VEL
LIN {X 0,Y 559.296,Z 363.647,A -85,B 0,C 180,E1 -2960.233,E2 -2960.233} C_VEL
LIN {X 0,Y 559.134,Z 372.786,A -85,B 0,C 180,E1 -2961.143,E2 -2961.143} C_VEL
LIN {X 0,Y 559.009,Z 381.688,A -85,B 0,C 180,E1 -2962.233,E2 -2962.233} C_VEL
LIN {X 0,Y 558.925,Z 387.74,A -85,B 0,C 180,E1 -2963.14,E2 -2963.14} C_VEL
LIN {X 0,Y 558.936,Z 393.68,A -85,B 0,C 180,E1 -2964.227,E2 -2964.227} C_VEL
LIN {X 0,Y 558.826,Z 398.373,A -85,B 0,C 180,E1 -2965.311,E2 -2965.311} C_VEL
LIN {X 0,Y 558.836,Z 401.958,A -85,B 0,C 180,E1 -2966.395,E2 -2966.395} C_VEL
LIN {X 0,Y 558.799,Z 403.807,A -85,B 0,C 180,E1 -2967.116,E2 -2967.116} C_VEL
LIN {X 0,Y 558.745,Z 406.183,A -85,B 0,C 180,E1 -2968.559,E2 -2968.559} C_VEL
LIN {X 0,Y 558.74,Z 407,A -85,B 0,C 180,E1 -2970,E2 -2970} C_VEL
LIN {X 0,Y 558.745,Z 406.184,A -85,B 0,C 180,E1 -2971.442,E2 -2971.442} C_VEL
LIN {X 0,Y 558.799,Z 403.81,A -85,B 0,C 180,E1 -2972.884,E2 -2972.884} C_VEL
LIN {X 0,Y 558.844,Z 400.895,A -85,B 0,C 180,E1 -2973.966,E2 -2973.966} C_VEL
LIN {X 0,Y 558.798,Z 396.948,A -85,B 0,C 180,E1 -2975.051,E2 -2975.051} C_VEL
LIN {X 0,Y 558.922,Z 391.867,A -85,B 0,C 180,E1 -2976.136,E2 -2976.136} C_VEL
LIN {X 0,Y 558.977,Z 385.467,A -85,B 0,C 180,E1 -2977.223,E2 -2977.223} C_VEL
LIN {X 0,Y 559.099,Z 377.477,A -85,B 0,C 180,E1 -2978.312,E2 -2978.312} C_VEL
LIN {X 0,Y 559.195,Z 369.333,A -85,B 0,C 180,E1 -2979.221,E2 -2979.221} C_VEL
LIN {X 0,Y 559.357,Z 359.397,A -85,B 0,C 180,E1 -2980.131,E2 -2980.131} C_VEL
LIN {X 0,Y 559.556,Z 348.397,A -85,B 0,C 180,E1 -2980.937,E2 -2980.937} C_VEL
LIN {X 0,Y 559.671,Z 336.457,A -85,B 0,C 180,E1 -2981.628,E2 -2981.628} C_VEL
LIN {X 0,Y 559.797,Z 324.976,A -85,B 0,C 180,E1 -2982.139,E2 -2982.139} C_VEL
LIN {X 0,Y 559.955,Z 312.173,A -85,B 0,C 180,E1 -2982.55,E2 -2982.55} C_VEL
LIN {X 0,Y 560.108,Z 298.596,A -85,B 0,C 180,E1 -2982.823,E2 -2982.823} C_VEL
LIN {X 0,Y 560.201,Z 200.442,A -85,B 0,C 180,E1 -2984.091,E2 -2984.091} C_VEL
LIN {X 0,Y 559.365,Z 194.797,A -85,B 0,C 180,E1 -2984.205,E2 -2984.205} C_VEL
LIN {X 0,Y 559.569,Z 173.746,A -85,B 0,C 180,E1 -2987.343,E2 -2987.343} C_VEL
LIN {X 0,Y 559.886,Z 153.609,A -85,B 0,C 180,E1 -2990.385,E2 -2990.385} C_VEL
LIN {X 0,Y 559.969,Z 141.061,A -85,B 0,C 180,E1 -2992.312,E2 -2992.312} C_VEL
LIN {X 0,Y 559.134,Z 136.341,A -85,B 0,C 180,E1 -2993.113,E2 -2993.113} C_VEL
LIN {X 0,Y 559.159,Z 136.33,A -85,B 0,C 180,E1 -2996.098,E2 -2996.098} C_VEL
LIN {X 0,Y 559.11,Z 136.336,A -85,B 0,C 180,E1 -2998.533,E2 -2998.533} C_VEL
LIN {X 0,Y 559.138,Z 136.336,A -85,B 0,C 180,E1 -3001.271,E2 -3001.271} C_VEL
LIN {X 0,Y 559.154,Z 136.329,A -85,B 0,C 180,E1 -3003.947,E2 -3003.947} C_VEL
LIN {X 0,Y 559.14,Z 136.336,A -85,B 0,C 180,E1 -3007.108,E2 -3007.108} C_VEL
LIN {X 0,Y 559.157,Z 136.329,A -85,B 0,C 180,E1 -3009.941,E2 -3009.941} C_VEL
LIN {X 0,Y 559.15,Z 136.337,A -85,B 0,C 180,E1 -3012.744,E2 -3012.744} C_VEL
LIN {X 0,Y 559.147,Z 136.33,A -85,B 0,C 180,E1 -3015.761,E2 -3015.761} C_VEL
LIN {X 0,Y 559.155,Z 136.334,A -85,B 0,C 180,E1 -3018.229,E2 -3018.229} C_VEL
LIN {X 0,Y 559.174,Z 136.327,A -85,B 0,C 180,E1 -3021.192,E2 -3021.192} C_VEL
LIN {X 0,Y 559.121,Z 136.335,A -85,B 0,C 180,E1 -3023.788,E2 -3023.788} C_VEL
LIN {X 0,Y 559.162,Z 136.334,A -85,B 0,C 180,E1 -3026.425,E2 -3026.425} C_VEL
LIN {X 0,Y 559.149,Z 136.33,A -85,B 0,C 180,E1 -3028.98,E2 -3028.98} C_VEL
LIN {X 0,Y 559.144,Z 136.333,A -85,B 0,C 180,E1 -3031.623,E2 -3031.623} C_VEL
LIN {X 0,Y 559.163,Z 136.336,A -85,B 0,C 180,E1 -3033.902,E2 -3033.902} C_VEL
LIN {X 0,Y 559.139,Z 136.332,A -85,B 0,C 180,E1 -3036.572,E2 -3036.572} C_VEL
LIN {X 0,Y 559.174,Z 136.329,A -85,B 0,C 180,E1 -3039.395,E2 -3039.395} C_VEL
LIN {X 0,Y 559.138,Z 136.339,A -85,B 0,C 180,E1 -3041.685,E2 -3041.685} C_VEL
LIN {X 0,Y 559.16,Z 136.334,A -85,B 0,C 180,E1 -3043.948,E2 -3043.948} C_VEL
LIN {X 0,Y 559.169,Z 136.329,A -85,B 0,C 180,E1 -3046.184,E2 -3046.184} C_VEL
LIN {X 0,Y 559.195,Z 136.327,A -85,B 0,C 180,E1 -3049.134,E2 -3049.134} C_VEL
LIN {X 0,Y 559.199,Z 136.325,A -85,B 0,C 180,E1 -3052.054,E2 -3052.054} C_VEL
LIN {X 0,Y 559.254,Z 136.32,A -85,B 0,C 180,E1 -3054.953,E2 -3054.953} C_VEL
LIN {X 0,Y 559.257,Z 136.318,A -85,B 0,C 180,E1 -3057.839,E2 -3057.839} C_VEL
LIN {X 0,Y 559.267,Z 136.317,A -85,B 0,C 180,E1 -3060.72,E2 -3060.72} C_VEL
LIN {X 0,Y 559.234,Z 136.324,A -85,B 0,C 180,E1 -3062.881,E2 -3062.881} C_VEL
LIN {X 0,Y 559.232,Z 136.32,A -85,B 0,C 180,E1 -3065.77,E2 -3065.77} C_VEL
LIN {X 0,Y 559.185,Z 136.33,A -85,B 0,C 180,E1 -3068.674,E2 -3068.674} C_VEL
LIN {X 0,Y 559.205,Z 136.323,A -85,B 0,C 180,E1 -3071.601,E2 -3071.601} C_VEL
LIN {X 0,Y 559.2,Z 136.33,A -85,B 0,C 180,E1 -3074.596,E2 -3074.596} C_VEL
LIN {X 0,Y 559.159,Z 136.329,A -85,B 0,C 180,E1 -3077.557,E2 -3077.557} C_VEL
LIN {X 0,Y 559.172,Z 136.327,A -85,B 0,C 180,E1 -3079.837,E2 -3079.837} C_VEL
LIN {X 0,Y 559.142,Z 136.334,A -85,B 0,C 180,E1 -3082.153,E2 -3082.153} C_VEL
LIN {X 0,Y 559.176,Z 136.326,A -85,B 0,C 180,E1 -3085.298,E2 -3085.298} C_VEL
LIN {X 0,Y 559.158,Z 136.329,A -85,B 0,C 180,E1 -3087.714,E2 -3087.714} C_VEL
LIN {X 0,Y 559.14,Z 136.333,A -85,B 0,C 180,E1 -3090.605,E2 -3090.605} C_VEL
LIN {X 0,Y 558.478,Z 136.416,A -85,B 0,C 180,E1 -3091.206,E2 -3091.206} C_VEL
LIN {X 0,Y 555.616,Z 136.778,A -85,B 0,C 180,E1 -3092.182,E2 -3092.182} C_VEL
LIN {X 0,Y 553.204,Z 137.073,A -85,B 0,C 180,E1 -3092.968,E2 -3092.968} C_VEL
LIN {X 0,Y 552.184,Z 137.199,A -85,B 0,C 180,E1 -3093.575,E2 -3093.575} C_VEL
LIN {X 0,Y 552.11,Z 137.21,A -85,B 0,C 180,E1 -3093.78,E2 -3093.78} C_VEL
LIN {X 0,Y 552.106,Z 137.208,A -85,B 0,C 180,E1 -3096.747,E2 -3096.747} C_VEL
LIN {X 0,Y 552.133,Z 137.206,A -85,B 0,C 180,E1 -3099.527,E2 -3099.527} C_VEL
LIN {X 0,Y 552.132,Z 137.207,A -85,B 0,C 180,E1 -3102.426,E2 -3102.426} C_VEL
LIN {X 0,Y 552.099,Z 137.212,A -85,B 0,C 180,E1 -3105.563,E2 -3105.563} C_VEL
LIN {X 0,Y 552.132,Z 137.204,A -85,B 0,C 180,E1 -3108.555,E2 -3108.555} C_VEL
LIN {X 0,Y 552.119,Z 137.21,A -85,B 0,C 180,E1 -3111.411,E2 -3111.411} C_VEL
LIN {X 0,Y 552.087,Z 137.211,A -85,B 0,C 180,E1 -3114.157,E2 -3114.157} C_VEL
LIN {X 0,Y 552.109,Z 137.207,A -85,B 0,C 180,E1 -3116.814,E2 -3116.814} C_VEL
LIN {X 0,Y 552.102,Z 137.216,A -85,B 0,C 180,E1 -3119.391,E2 -3119.391} C_VEL
LIN {X 0,Y 552.108,Z 137.209,A -85,B 0,C 180,E1 -3121.902,E2 -3121.902} C_VEL
LIN {X 0,Y 552.158,Z 137.203,A -85,B 0,C 180,E1 -3124.65,E2 -3124.65} C_VEL
LIN {X 0,Y 552.094,Z 137.215,A -85,B 0,C 180,E1 -3127.549,E2 -3127.549} C_VEL
LIN {X 0,Y 552.172,Z 137.354,A -85,B 0,C 180,E1 -3129.658,E2 -3129.658} C_VEL
LIN {X 0,Y 552.614,Z 141.77,A -85,B 0,C 180,E1 -3130.466,E2 -3130.466} C_VEL
LIN {X 0,Y 552.451,Z 155.952,A -85,B 0,C 180,E1 -3132.987,E2 -3132.987} C_VEL
LIN {X 0,Y 552.253,Z 171.292,A -85,B 0,C 180,E1 -3135.686,E2 -3135.686} C_VEL
LIN {X 0,Y 553.458,Z 179.269,A -85,B 0,C 180,E1 -3135.825,E2 -3135.825} C_VEL
LIN {X 0,Y 553.133,Z 278.233,A -85,B 0,C 180,E1 -3137.129,E2 -3137.129} C_VEL
LIN {X 0,Y 552.996,Z 291.454,A -85,B 0,C 180,E1 -3137.453,E2 -3137.453} C_VEL
LIN {X 0,Y 552.84,Z 303.575,A -85,B 0,C 180,E1 -3137.892,E2 -3137.892} C_VEL
LIN {X 0,Y 552.688,Z 315.062,A -85,B 0,C 180,E1 -3138.451,E2 -3138.451} C_VEL
LIN {X 0,Y 552.496,Z 326.696,A -85,B 0,C 180,E1 -3139.186,E2 -3139.186} C_VEL
LIN {X 0,Y 552.305,Z 337.184,A -85,B 0,C 180,E1 -3140.016,E2 -3140.016} C_VEL
LIN {X 0,Y 552.178,Z 345.753,A -85,B 0,C 180,E1 -3140.846,E2 -3140.846} C_VEL
LIN {X 0,Y 552.007,Z 353.646,A -85,B 0,C 180,E1 -3141.765,E2 -3141.765} C_VEL
LIN {X 0,Y 551.895,Z 361.477,A -85,B 0,C 180,E1 -3142.886,E2 -3142.886} C_VEL
LIN {X 0,Y 551.868,Z 368.456,A -85,B 0,C 180,E1 -3144.153,E2 -3144.153} C_VEL
LIN {X 0,Y 551.725,Z 373.197,A -85,B 0,C 180,E1 -3145.251,E2 -3145.251} C_VEL
LIN {X 0,Y 551.751,Z 376.829,A -85,B 0,C 180,E1 -3146.348,E2 -3146.348} C_VEL
LIN {X 0,Y 551.723,Z 378.707,A -85,B 0,C 180,E1 -3147.079,E2 -3147.079} C_VEL
LIN {X 0,Y 551.657,Z 380.126,A -85,B 0,C 180,E1 -3147.81,E2 -3147.81} C_VEL
LIN {X 0,Y 551.642,Z 381.756,A -85,B 0,C 180,E1 -3149.27,E2 -3149.27} C_VEL
LIN {X 0,Y 551.641,Z 381.996,A -85,B 0,C 180,E1 -3150,E2 -3150} C_VEL
LIN {X 0,Y 551.641,Z 381.815,A -85,B 0,C 180,E1 -3150.73,E2 -3150.73} C_VEL
LIN {X 0,Y 551.657,Z 380.262,A -85,B 0,C 180,E1 -3152.19,E2 -3152.19} C_VEL
LIN {X 0,Y 551.724,Z 378.901,A -85,B 0,C 180,E1 -3152.921,E2 -3152.921} C_VEL
LIN {X 0,Y 551.764,Z 376.025,A -85,B 0,C 180,E1 -3154.017,E2 -3154.017} C_VEL
LIN {X 0,Y 551.723,Z 372.125,A -85,B 0,C 180,E1 -3155.116,E2 -3155.116} C_VEL
LIN {X 0,Y 551.811,Z 366.393,A -85,B 0,C 180,E1 -3156.349,E2 -3156.349} C_VEL
LIN {X 0,Y 551.925,Z 359.561,A -85,B 0,C 180,E1 -3157.5,E2 -3157.5} C_VEL
LIN {X 0,Y 552.063,Z 351.41,A -85,B 0,C 180,E1 -3158.603,E2 -3158.603} C_VEL
LIN {X 0,Y 552.197,Z 343.069,A -85,B 0,C 180,E1 -3159.524,E2 -3159.524} C_VEL
LIN {X 0,Y 552.427,Z 332.774,A -85,B 0,C 180,E1 -3160.445,E2 -3160.445} C_VEL
LIN {X 0,Y 552.567,Z 321.959,A -85,B 0,C 180,E1 -3161.224,E2 -3161.224} C_VEL
LIN {X 0,Y 552.744,Z 311.424,A -85,B 0,C 180,E1 -3161.831,E2 -3161.831} C_VEL
LIN {X 0,Y 552.901,Z 298.916,A -85,B 0,C 180,E1 -3162.386,E2 -3162.386} C_VEL
LIN {X 0,Y 553.072,Z 285.489,A -85,B 0,C 180,E1 -3162.802,E2 -3162.802} C_VEL
LIN {X 0,Y 553.235,Z 272.178,A -85,B 0,C 180,E1 -3163.055,E2 -3163.055} C_VEL
LIN {X 0,Y 553.347,Z 177.516,A -85,B 0,C 180,E1 -3164.291,E2 -3164.291} C_VEL
LIN {X 0,Y 552.251,Z 171.162,A -85,B 0,C 180,E1 -3164.424,E2 -3164.424} C_VEL
LIN {X 0,Y 552.446,Z 154.82,A -85,B 0,C 180,E1 -3167.304,E2 -3167.304} C_VEL
LIN {X 0,Y 552.603,Z 141.03,A -85,B 0,C 180,E1 -3169.757,E2 -3169.757} C_VEL
LIN {X 0,Y 552.132,Z 137.212,A -85,B 0,C 180,E1 -3170.49,E2 -3170.49} C_VEL
LIN {X 0,Y 552.098,Z 137.21,A -85,B 0,C 180,E1 -3173.575,E2 -3173.575} C_VEL
LIN {X 0,Y 552.131,Z 137.205,A -85,B 0,C 180,E1 -3175.644,E2 -3175.644} C_VEL
LIN {X 0,Y 552.126,Z 137.212,A -85,B 0,C 180,E1 -3178.562,E2 -3178.562} C_VEL
LIN {X 0,Y 552.113,Z 137.206,A -85,B 0,C 180,E1 -3181.475,E2 -3181.475} C_VEL
LIN {X 0,Y 552.127,Z 137.208,A -85,B 0,C 180,E1 -3184.169,E2 -3184.169} C_VEL
LIN {X 0,Y 552.106,Z 137.212,A -85,B 0,C 180,E1 -3186.747,E2 -3186.747} C_VEL
LIN {X 0,Y 552.131,Z 137.204,A -85,B 0,C 180,E1 -3189.527,E2 -3189.527} C_VEL
LIN {X 0,Y 552.132,Z 137.211,A -85,B 0,C 180,E1 -3192.425,E2 -3192.425} C_VEL
LIN {X 0,Y 552.099,Z 137.209,A -85,B 0,C 180,E1 -3195.562,E2 -3195.562} C_VEL
LIN {X 0,Y 552.133,Z 137.205,A -85,B 0,C 180,E1 -3198.677,E2 -3198.677} C_VEL
LIN {X 0,Y 552.121,Z 137.207,A -85,B 0,C 180,E1 -3201.411,E2 -3201.411} C_VEL
LIN {X 0,Y 552.085,Z 137.215,A -85,B 0,C 180,E1 -3204.156,E2 -3204.156} C_VEL
LIN {X 0,Y 552.115,Z 137.206,A -85,B 0,C 180,E1 -3206.814,E2 -3206.814} C_VEL
LIN {X 0,Y 552.102,Z 137.211,A -85,B 0,C 180,E1 -3209.391,E2 -3209.391} C_VEL
LIN {X 0,Y 552.11,Z 137.212,A -85,B 0,C 180,E1 -3211.902,E2 -3211.902} C_VEL
LIN {X 0,Y 552.156,Z 137.201,A -85,B 0,C 180,E1 -3214.649,E2 -3214.649} C_VEL
LIN {X 0,Y 552.093,Z 137.217,A -85,B 0,C 180,E1 -3217.549,E2 -3217.549} C_VEL
LIN {X 0,Y 552.149,Z 137.202,A -85,B 0,C 180,E1 -3220.373,E2 -3220.373} C_VEL
LIN {X 0,Y 552.155,Z 137.205,A -85,B 0,C 180,E1 -3222.977,E2 -3222.977} C_VEL
LIN {X 0,Y 552.135,Z 137.204,A -85,B 0,C 180,E1 -3226.004,E2 -3226.004} C_VEL
LIN {X 0,Y 552.162,Z 137.207,A -85,B 0,C 180,E1 -3228.993,E2 -3228.993} C_VEL
LIN {X 0,Y 552.157,Z 137.201,A -85,B 0,C 180,E1 -3231.951,E2 -3231.951} C_VEL
LIN {X 0,Y 552.227,Z 137.2,A -85,B 0,C 180,E1 -3234.889,E2 -3234.889} C_VEL
LIN {X 0,Y 552.226,Z 137.192,A -85,B 0,C 180,E1 -3237.812,E2 -3237.812} C_VEL
LIN {X 0,Y 552.244,Z 137.198,A -85,B 0,C 180,E1 -3240.729,E2 -3240.729} C_VEL
LIN {X 0,Y 552.203,Z 137.201,A -85,B 0,C 180,E1 -3242.918,E2 -3242.918} C_VEL
LIN {X 0,Y 552.2,Z 137.196,A -85,B 0,C 180,E1 -3245.844,E2 -3245.844} C_VEL
LIN {X 0,Y 552.153,Z 137.207,A -85,B 0,C 180,E1 -3248.786,E2 -3248.786} C_VEL
LIN {X 0,Y 552.161,Z 137.201,A -85,B 0,C 180,E1 -3251.751,E2 -3251.751} C_VEL
LIN {X 0,Y 552.135,Z 137.207,A -85,B 0,C 180,E1 -3254.748,E2 -3254.748} C_VEL
LIN {X 0,Y 552.097,Z 137.211,A -85,B 0,C 180,E1 -3257.789,E2 -3257.789} C_VEL
LIN {X 0,Y 552.125,Z 137.213,A -85,B 0,C 180,E1 -3260.101,E2 -3260.101} C_VEL
LIN {X 0,Y 552.091,Z 137.213,A -85,B 0,C 180,E1 -3262.451,E2 -3262.451} C_VEL
LIN {X 0,Y 552.136,Z 137.204,A -85,B 0,C 180,E1 -3265.346,E2 -3265.346} C_VEL
LIN {X 0,Y 552.088,Z 137.216,A -85,B 0,C 180,E1 -3268.1,E2 -3268.1} C_VEL
LIN {X 0,Y 552.099,Z 137.208,A -85,B 0,C 180,E1 -3270.61,E2 -3270.61} C_VEL
LIN {X 0,Y 552.114,Z 137.207,A -85,B 0,C 180,E1 -3273.186,E2 -3273.186} C_VEL
LIN {X 0,Y 552.074,Z 137.219,A -85,B 0,C 180,E1 -3275.845,E2 -3275.845} C_VEL
LIN {X 0,Y 552.116,Z 137.206,A -85,B 0,C 180,E1 -3278.589,E2 -3278.589} C_VEL
LIN {X 0,Y 552.11,Z 137.214,A -85,B 0,C 180,E1 -3281.447,E2 -3281.447} C_VEL
LIN {X 0,Y 552.088,Z 137.209,A -85,B 0,C 180,E1 -3284.531,E2 -3284.531} C_VEL
LIN {X 0,Y 552.109,Z 137.213,A -85,B 0,C 180,E1 -3287.587,E2 -3287.587} C_VEL
LIN {X 0,Y 552.127,Z 137.205,A -85,B 0,C 180,E1 -3290.473,E2 -3290.473} C_VEL
LIN {X 0,Y 552.106,Z 137.214,A -85,B 0,C 180,E1 -3293.317,E2 -3293.317} C_VEL
LIN {X 0,Y 552.1,Z 137.208,A -85,B 0,C 180,E1 -3295.937,E2 -3295.937} C_VEL
LIN {X 0,Y 552.104,Z 137.21,A -85,B 0,C 180,E1 -3298.54,E2 -3298.54} C_VEL
LIN {X 0,Y 552.08,Z 137.213,A -85,B 0,C 180,E1 -3301.447,E2 -3301.447} C_VEL
LIN {X 0,Y 552.083,Z 137.214,A -85,B 0,C 180,E1 -3304.354,E2 -3304.354} C_VEL
LIN {X 0,Y 552.118,Z 137.284,A -85,B 0,C 180,E1 -3306.784,E2 -3306.784} C_VEL
LIN {X 0,Y 552.996,Z 142.166,A -85,B 0,C 180,E1 -3307.588,E2 -3307.588} C_VEL
LIN {X 0,Y 552.784,Z 158.945,A -85,B 0,C 180,E1 -3310.191,E2 -3310.191} C_VEL
LIN {X 0,Y 552.524,Z 177.264,A -85,B 0,C 180,E1 -3312.989,E2 -3312.989} C_VEL
LIN {X 0,Y 552.337,Z 194.754,A -85,B 0,C 180,E1 -3315.628,E2 -3315.628} C_VEL
LIN {X 0,Y 553.392,Z 202.717,A -85,B 0,C 180,E1 -3315.764,E2 -3315.764} C_VEL
LIN {X 0,Y 553.13,Z 302.787,A -85,B 0,C 180,E1 -3317.083,E2 -3317.083} C_VEL
LIN {X 0,Y 552.973,Z 316.069,A -85,B 0,C 180,E1 -3317.406,E2 -3317.406} C_VEL
LIN {X 0,Y 552.802,Z 329.36,A -85,B 0,C 180,E1 -3317.891,E2 -3317.891} C_VEL
LIN {X 0,Y 552.63,Z 341.092,A -85,B 0,C 180,E1 -3318.48,E2 -3318.48} C_VEL
LIN {X 0,Y 552.446,Z 353.407,A -85,B 0,C 180,E1 -3319.278,E2 -3319.278} C_VEL
LIN {X 0,Y 552.283,Z 363.599,A -85,B 0,C 180,E1 -3320.108,E2 -3320.108} C_VEL
LIN {X 0,Y 552.104,Z 372.768,A -85,B 0,C 180,E1 -3321.029,E2 -3321.029} C_VEL
LIN {X 0,Y 551.96,Z 381.688,A -85,B 0,C 180,E1 -3322.133,E2 -3322.133} C_VEL
LIN {X 0,Y 551.835,Z 388.849,A -85,B 0,C 180,E1 -3323.235,E2 -3323.235} C_VEL
LIN {X 0,Y 551.804,Z 395.366,A -85,B 0,C 180,E1 -3324.519,E2 -3324.519} C_VEL
LIN {X 0,Y 551.764,Z 399.677,A -85,B 0,C 180,E1 -3325.617,E2 -3325.617} C_VEL
LIN {X 0,Y 551.75,Z 401.958,A -85,B 0,C 180,E1 -3326.349,E2 -3326.349} C_VEL
LIN {X 0,Y 551.723,Z 403.807,A -85,B 0,C 180,E1 -3327.079,E2 -3327.079} C_VEL
LIN {X 0,Y 551.645,Z 406.182,A -85,B 0,C 180,E1 -3328.54,E2 -3328.54} C_VEL
LIN {X 0,Y 551.64,Z 407,A -85,B 0,C 180,E1 -3330,E2 -3330} C_VEL
LIN {X 0,Y 551.645,Z 406.183,A -85,B 0,C 180,E1 -3331.46,E2 -3331.46} C_VEL
LIN {X 0,Y 551.723,Z 403.81,A -85,B 0,C 180,E1 -3332.921,E2 -3332.921} C_VEL
LIN {X 0,Y 551.764,Z 400.895,A -85,B 0,C 180,E1 -3334.017,E2 -3334.017} C_VEL
LIN {X 0,Y 551.723,Z 396.948,A -85,B 0,C 180,E1 -3335.116,E2 -3335.116} C_VEL
LIN {X 0,Y 551.803,Z 391.188,A -85,B 0,C 180,E1 -3336.342,E2 -3336.342} C_VEL
LIN {X 0,Y 551.926,Z 384.235,A -85,B 0,C 180,E1 -3337.5,E2 -3337.5} C_VEL
LIN {X 0,Y 552.082,Z 375.986,A -85,B 0,C 180,E1 -3338.602,E2 -3338.602} C_VEL
LIN {X 0,Y 552.2,Z 367.505,A -85,B 0,C 180,E1 -3339.524,E2 -3339.524} C_VEL
LIN {X 0,Y 552.428,Z 357.024,A -85,B 0,C 180,E1 -3340.445,E2 -3340.445} C_VEL
LIN {X 0,Y 552.575,Z 346.19,A -85,B 0,C 180,E1 -3341.214,E2 -3341.214} C_VEL
LIN {X 0,Y 552.752,Z 335.285,A -85,B 0,C 180,E1 -3341.831,E2 -3341.831} C_VEL
LIN {X 0,Y 552.922,Z 323.625,A -85,B 0,C 180,E1 -3342.339,E2 -3342.339} C_VEL
LIN {X 0,Y 553.017,Z 311.102,A -85,B 0,C 180,E1 -3342.733,E2 -3342.733} C_VEL
LIN {X 0,Y 553.205,Z 298.435,A -85,B 0,C 180,E1 -3342.985,E2 -3342.985} C_VEL
LIN {X 0,Y 553.228,Z 200.491,A -85,B 0,C 180,E1 -3344.269,E2 -3344.269} C_VEL
LIN {X 0,Y 552.358,Z 194.632,A -85,B 0,C 180,E1 -3344.389,E2 -3344.389} C_VEL
LIN {X 0,Y 552.568,Z 175.06,A -85,B 0,C 180,E1 -3347.345,E2 -3347.345} C_VEL
LIN {X 0,Y 552.932,Z 154.71,A -85,B 0,C 180,E1 -3350.459,E2 -3350.459} C_VEL
LIN {X 0,Y 552.996,Z 142.165,A -85,B 0,C 180,E1 -3352.412,E2 -3352.412} C_VEL
LIN {X 0,Y 552.102,Z 137.217,A -85,B 0,C 180,E1 -3353.242,E2 -3353.242} C_VEL
LIN {X 0,Y 552.095,Z 137.211,A -85,B 0,C 180,E1 -3356.458,E2 -3356.458} C_VEL
LIN {X 0,Y 552.05,Z 137.221,A -85,B 0,C 180,E1 -3358.932,E2 -3358.932} C_VEL
LIN {X 0,Y 552.092,Z 137.211,A -85,B 0,C 180,E1 -3361.472,E2 -3361.472} C_VEL
LIN {X 0,Y 552.123,Z 137.206,A -85,B 0,C 180,E1 -3364.168,E2 -3364.168} C_VEL
LIN {X 0,Y 552.105,Z 137.216,A -85,B 0,C 180,E1 -3366.747,E2 -3366.747} C_VEL
LIN {X 0,Y 552.126,Z 137.205,A -85,B 0,C 180,E1 -3369.527,E2 -3369.527} C_VEL
LIN {X 0,Y 552.109,Z 137.213,A -85,B 0,C 180,E1 -3372.427,E2 -3372.427} C_VEL
LIN {X 0,Y 552.091,Z 137.209,A -85,B 0,C 180,E1 -3375.562,E2 -3375.562} C_VEL
LIN {X 0,Y 552.108,Z 137.213,A -85,B 0,C 180,E1 -3378.68,E2 -3378.68} C_VEL
LIN {X 0,Y 552.116,Z 137.206,A -85,B 0,C 180,E1 -3381.411,E2 -3381.411} C_VEL
LIN {X 0,Y 552.074,Z 137.218,A -85,B 0,C 180,E1 -3384.155,E2 -3384.155} C_VEL
LIN {X 0,Y 552.114,Z 137.208,A -85,B 0,C 180,E1 -3386.814,E2 -3386.814} C_VEL
LIN {X 0,Y 552.096,Z 137.209,A -85,B 0,C 180,E1 -3389.39,E2 -3389.39} C_VEL
LIN {X 0,Y 552.087,Z 137.216,A -85,B 0,C 180,E1 -3391.9,E2 -3391.9} C_VEL
LIN {X 0,Y 552.136,Z 137.204,A -85,B 0,C 180,E1 -3394.654,E2 -3394.654} C_VEL
LIN {X 0,Y 552.091,Z 137.213,A -85,B 0,C 180,E1 -3397.549,E2 -3397.549} C_VEL
LIN {X 0,Y 552.144,Z 137.204,A -85,B 0,C 180,E1 -3400.375,E2 -3400.375} C_VEL
LIN {X 0,Y 552.132,Z 137.204,A -85,B 0,C 180,E1 -3402.977,E2 -3402.977} C_VEL
LIN {X 0,Y 552.133,Z 137.208,A -85,B 0,C 180,E1 -3406.004,E2 -3406.004} C_VEL
LIN {X 0,Y 552.163,Z 137.202,A -85,B 0,C 180,E1 -3408.993,E2 -3408.993} C_VEL
LIN {X 0,Y 552.154,Z 137.204,A -85,B 0,C 180,E1 -3411.951,E2 -3411.951} C_VEL
LIN {X 0,Y 552.229,Z 137.194,A -85,B 0,C 180,E1 -3414.889,E2 -3414.889} C_VEL
LIN {X 0,Y 552.228,Z 137.194,A -85,B 0,C 180,E1 -3417.812,E2 -3417.812} C_VEL
LIN {X 0,Y 552.238,Z 137.193,A -85,B 0,C 180,E1 -3420.729,E2 -3420.729} C_VEL
LIN {X 0,Y 552.202,Z 137.201,A -85,B 0,C 180,E1 -3422.918,E2 -3422.918} C_VEL
LIN {X 0,Y 552.201,Z 137.196,A -85,B 0,C 180,E1 -3425.844,E2 -3425.844} C_VEL
LIN {X 0,Y 552.153,Z 137.208,A -85,B 0,C 180,E1 -3428.786,E2 -3428.786} C_VEL
LIN {X 0,Y 552.163,Z 137.2,A -85,B 0,C 180,E1 -3431.751,E2 -3431.751} C_VEL
LIN {X 0,Y 552.137,Z 137.212,A -85,B 0,C 180,E1 -3434.748,E2 -3434.748} C_VEL
LIN {X 0,Y 552.11,Z 137.206,A -85,B 0,C 180,E1 -3437.789,E2 -3437.789} C_VEL
LIN {X 0,Y 552.131,Z 137.206,A -85,B 0,C 180,E1 -3440.101,E2 -3440.101} C_VEL
LIN {X 0,Y 552.094,Z 137.216,A -85,B 0,C 180,E1 -3442.451,E2 -3442.451} C_VEL
LIN {X 0,Y 552.156,Z 137.201,A -85,B 0,C 180,E1 -3445.351,E2 -3445.351} C_VEL
LIN {X 0,Y 552.11,Z 137.211,A -85,B 0,C 180,E1 -3448.098,E2 -3448.098} C_VEL
LIN {X 0,Y 552.103,Z 137.212,A -85,B 0,C 180,E1 -3450.609,E2 -3450.609} C_VEL
LIN {X 0,Y 552.116,Z 137.206,A -85,B 0,C 180,E1 -3453.186,E2 -3453.186} C_VEL
LIN {X 0,Y 552.11,Z 137.21,A -85,B 0,C 180,E1 -3453.78,E2 -3453.78} C_VEL
LIN {X 0,Y 551.474,Z 137.295,A -85,B 0,C 180,E1 -3454.389,E2 -3454.389} C_VEL
LIN {X 0,Y 548.653,Z 137.645,A -85,B 0,C 180,E1 -3455.377,E2 -3455.377} C_VEL
LIN {X 0,Y 546.233,Z 137.948,A -85,B 0,C 180,E1 -3456.172,E2 -3456.172} C_VEL
LIN {X 0,Y 545.165,Z 138.073,A -85,B 0,C 180,E1 -3456.786,E2 -3456.786} C_VEL
LIN {X 0,Y 545.063,Z 138.084,A -85,B 0,C 180,E1 -3456.994,E2 -3456.994} C_VEL
LIN {X 0,Y 545.073,Z 138.091,A -85,B 0,C 180,E1 -3460.142,E2 -3460.142} C_VEL
LIN {X 0,Y 545.08,Z 138.083,A -85,B 0,C 180,E1 -3463.107,E2 -3463.107} C_VEL
LIN {X 0,Y 545.069,Z 138.087,A -85,B 0,C 180,E1 -3466.224,E2 -3466.224} C_VEL
LIN {X 0,Y 545.088,Z 138.081,A -85,B 0,C 180,E1 -3468.886,E2 -3468.886} C_VEL
LIN {X 0,Y 545.054,Z 138.094,A -85,B 0,C 180,E1 -3471.763,E2 -3471.763} C_VEL
LIN {X 0,Y 545.038,Z 138.088,A -85,B 0,C 180,E1 -3474.532,E2 -3474.532} C_VEL
LIN {X 0,Y 545.067,Z 138.088,A -85,B 0,C 180,E1 -3477.212,E2 -3477.212} C_VEL
LIN {X 0,Y 545.063,Z 138.088,A -85,B 0,C 180,E1 -3479.811,E2 -3479.811} C_VEL
LIN {X 0,Y 545.08,Z 138.082,A -85,B 0,C 180,E1 -3482.344,E2 -3482.344} C_VEL
LIN {X 0,Y 545.12,Z 138.081,A -85,B 0,C 180,E1 -3484.821,E2 -3484.821} C_VEL
LIN {X 0,Y 545.039,Z 138.096,A -85,B 0,C 180,E1 -3487.242,E2 -3487.242} C_VEL
LIN {X 0,Y 545.124,Z 138.179,A -85,B 0,C 180,E1 -3489.531,E2 -3489.531} C_VEL
LIN {X 0,Y 545.623,Z 143.041,A -85,B 0,C 180,E1 -3490.434,E2 -3490.434} C_VEL
LIN {X 0,Y 545.447,Z 155.994,A -85,B 0,C 180,E1 -3492.761,E2 -3492.761} C_VEL
LIN {X 0,Y 545.244,Z 171.374,A -85,B 0,C 180,E1 -3495.491,E2 -3495.491} C_VEL
LIN {X 0,Y 546.601,Z 179.608,A -85,B 0,C 180,E1 -3495.645,E2 -3495.645} C_VEL
LIN {X 0,Y 546.217,Z 278.424,A -85,B 0,C 180,E1 -3496.964,E2 -3496.964} C_VEL
LIN {X 0,Y 546.078,Z 291.635,A -85,B 0,C 180,E1 -3497.291,E2 -3497.291} C_VEL
LIN {X 0,Y 545.901,Z 303.752,A -85,B 0,C 180,E1 -3497.736,E2 -3497.736} C_VEL
LIN {X 0,Y 545.727,Z 315.938,A -85,B 0,C 180,E1 -3498.342,E2 -3498.342} C_VEL
LIN {X 0,Y 545.529,Z 326.866,A -85,B 0,C 180,E1 -3499.046,E2 -3499.046} C_VEL
LIN {X 0,Y 545.3,Z 337.354,A -85,B 0,C 180,E1 -3499.886,E2 -3499.886} C_VEL
LIN {X 0,Y 545.157,Z 345.921,A -85,B 0,C 180,E1 -3500.727,E2 -3500.727} C_VEL
LIN {X 0,Y 544.975,Z 353.814,A -85,B 0,C 180,E1 -3501.658,E2 -3501.658} C_VEL
LIN {X 0,Y 544.83,Z 361.533,A -85,B 0,C 180,E1 -3502.775,E2 -3502.775} C_VEL
LIN {X 0,Y 544.801,Z 368.608,A -85,B 0,C 180,E1 -3504.076,E2 -3504.076} C_VEL
LIN {X 0,Y 544.633,Z 373.329,A -85,B 0,C 180,E1 -3505.189,E2 -3505.189} C_VEL
LIN {X 0,Y 544.669,Z 376.942,A -85,B 0,C 180,E1 -3506.301,E2 -3506.301} C_VEL
LIN {X 0,Y 544.65,Z 378.811,A -85,B 0,C 180,E1 -3507.041,E2 -3507.041} C_VEL
LIN {X 0,Y 544.572,Z 380.224,A -85,B 0,C 180,E1 -3507.781,E2 -3507.781} C_VEL
LIN {X 0,Y 544.543,Z 381.845,A -85,B 0,C 180,E1 -3509.26,E2 -3509.26} C_VEL
LIN {X 0,Y 544.542,Z 382.084,A -85,B 0,C 180,E1 -3510,E2 -3510} C_VEL
LIN {X 0,Y 544.542,Z 381.903,A -85,B 0,C 180,E1 -3510.739,E2 -3510.739} C_VEL
LIN {X 0,Y 544.572,Z 380.357,A -85,B 0,C 180,E1 -3512.219,E2 -3512.219} C_VEL
LIN {X 0,Y 544.651,Z 379.001,A -85,B 0,C 180,E1 -3512.959,E2 -3512.959} C_VEL
LIN {X 0,Y 544.684,Z 376.139,A -85,B 0,C 180,E1 -3514.069,E2 -3514.069} C_VEL
LIN {X 0,Y 544.653,Z 372.257,A -85,B 0,C 180,E1 -3515.182,E2 -3515.182} C_VEL
LIN {X 0,Y 544.748,Z 367.055,A -85,B 0,C 180,E1 -3516.335,E2 -3516.335} C_VEL
LIN {X 0,Y 544.878,Z 359.719,A -85,B 0,C 180,E1 -3517.597,E2 -3517.597} C_VEL
LIN {X 0,Y 545.036,Z 351.568,A -85,B 0,C 180,E1 -3518.714,E2 -3518.714} C_VEL
LIN {X 0,Y 545.183,Z 343.226,A -85,B 0,C 180,E1 -3519.647,E2 -3519.647} C_VEL
LIN {X 0,Y 545.424,Z 332.929,A -85,B 0,C 180,E1 -3520.58,E2 -3520.58} C_VEL
LIN {X 0,Y 545.627,Z 321.36,A -85,B 0,C 180,E1 -3521.419,E2 -3521.419} C_VEL
LIN {X 0,Y 545.855,Z 309.766,A -85,B 0,C 180,E1 -3522.077,E2 -3522.077} C_VEL
LIN {X 0,Y 546.044,Z 297.762,A -85,B 0,C 180,E1 -3522.591,E2 -3522.591} C_VEL
LIN {X 0,Y 546.169,Z 284.713,A -85,B 0,C 180,E1 -3522.99,E2 -3522.99} C_VEL
LIN {X 0,Y 546.328,Z 272.296,A -85,B 0,C 180,E1 -3523.223,E2 -3523.223} C_VEL
LIN {X 0,Y 546.48,Z 178.327,A -85,B 0,C 180,E1 -3524.466,E2 -3524.466} C_VEL
LIN {X 0,Y 545.257,Z 171.412,A -85,B 0,C 180,E1 -3524.592,E2 -3524.592} C_VEL
LIN {X 0,Y 545.492,Z 153.828,A -85,B 0,C 180,E1 -3527.716,E2 -3527.716} C_VEL
LIN {X 0,Y 545.607,Z 141.733,A -85,B 0,C 180,E1 -3529.894,E2 -3529.894} C_VEL
LIN {X 0,Y 545.087,Z 138.09,A -85,B 0,C 180,E1 -3530.619,E2 -3530.619} C_VEL
LIN {X 0,Y 545.055,Z 138.087,A -85,B 0,C 180,E1 -3533.725,E2 -3533.725} C_VEL
LIN {X 0,Y 545.081,Z 138.084,A -85,B 0,C 180,E1 -3536,E2 -3536} C_VEL
LIN {X 0,Y 545.091,Z 138.089,A -85,B 0,C 180,E1 -3538.748,E2 -3538.748} C_VEL
LIN {X 0,Y 545.056,Z 138.086,A -85,B 0,C 180,E1 -3541.915,E2 -3541.915} C_VEL
LIN {X 0,Y 545.061,Z 138.093,A -85,B 0,C 180,E1 -3544.564,E2 -3544.564} C_VEL
LIN {X 0,Y 545.037,Z 138.088,A -85,B 0,C 180,E1 -3547.304,E2 -3547.304} C_VEL
LIN {X 0,Y 545.067,Z 138.09,A -85,B 0,C 180,E1 -3550.142,E2 -3550.142} C_VEL
LIN {X 0,Y 545.079,Z 138.082,A -85,B 0,C 180,E1 -3553.106,E2 -3553.106} C_VEL
LIN {X 0,Y 545.068,Z 138.092,A -85,B 0,C 180,E1 -3556.224,E2 -3556.224} C_VEL
LIN {X 0,Y 545.092,Z 138.081,A -85,B 0,C 180,E1 -3558.886,E2 -3558.886} C_VEL
LIN {X 0,Y 545.055,Z 138.091,A -85,B 0,C 180,E1 -3561.763,E2 -3561.763} C_VEL
LIN {X 0,Y 545.036,Z 138.089,A -85,B 0,C 180,E1 -3564.531,E2 -3564.531} C_VEL
LIN {X 0,Y 545.069,Z 138.085,A -85,B 0,C 180,E1 -3567.211,E2 -3567.211} C_VEL
LIN {X 0,Y 545.064,Z 138.093,A -85,B 0,C 180,E1 -3569.81,E2 -3569.81} C_VEL
LIN {X 0,Y 545.081,Z 138.083,A -85,B 0,C 180,E1 -3572.344,E2 -3572.344} C_VEL
LIN {X 0,Y 545.117,Z 138.078,A -85,B 0,C 180,E1 -3574.82,E2 -3574.82} C_VEL
LIN {X 0,Y 545.038,Z 138.093,A -85,B 0,C 180,E1 -3577.242,E2 -3577.242} C_VEL
LIN {X 0,Y 545.12,Z 138.077,A -85,B 0,C 180,E1 -3580.415,E2 -3580.415} C_VEL
LIN {X 0,Y 545.073,Z 138.089,A -85,B 0,C 180,E1 -3583.521,E2 -3583.521} C_VEL
LIN {X 0,Y 545.094,Z 138.082,A -85,B 0,C 180,E1 -3585.82,E2 -3585.82} C_VEL
LIN {X 0,Y 545.118,Z 138.082,A -85,B 0,C 180,E1 -3588.849,E2 -3588.849} C_VEL
LIN {X 0,Y 545.128,Z 138.077,A -85,B 0,C 180,E1 -3591.847,E2 -3591.847} C_VEL
LIN {X 0,Y 545.203,Z 138.074,A -85,B 0,C 180,E1 -3594.823,E2 -3594.823} C_VEL
LIN {X 0,Y 545.197,Z 138.068,A -85,B 0,C 180,E1 -3597.784,E2 -3597.784} C_VEL
LIN {X 0,Y 545.214,Z 138.074,A -85,B 0,C 180,E1 -3600.739,E2 -3600.739} C_VEL
LIN {X 0,Y 545.17,Z 138.077,A -85,B 0,C 180,E1 -3602.956,E2 -3602.956} C_VEL
LIN {X 0,Y 545.171,Z 138.072,A -85,B 0,C 180,E1 -3605.919,E2 -3605.919} C_VEL
LIN {X 0,Y 545.11,Z 138.082,A -85,B 0,C 180,E1 -3608.9,E2 -3608.9} C_VEL
LIN {X 0,Y 545.134,Z 138.078,A -85,B 0,C 180,E1 -3611.904,E2 -3611.904} C_VEL
LIN {X 0,Y 545.084,Z 138.083,A -85,B 0,C 180,E1 -3614.944,E2 -3614.944} C_VEL
LIN {X 0,Y 545.069,Z 138.089,A -85,B 0,C 180,E1 -3618.026,E2 -3618.026} C_VEL
LIN {X 0,Y 545.091,Z 138.087,A -85,B 0,C 180,E1 -3620.372,E2 -3620.372} C_VEL
LIN {X 0,Y 545.078,Z 138.085,A -85,B 0,C 180,E1 -3623.56,E2 -3623.56} C_VEL
LIN {X 0,Y 545.074,Z 138.092,A -85,B 0,C 180,E1 -3626.001,E2 -3626.001} C_VEL
LIN {X 0,Y 545.073,Z 138.083,A -85,B 0,C 180,E1 -3628.745,E2 -3628.745} C_VEL
LIN {X 0,Y 545.057,Z 138.092,A -85,B 0,C 180,E1 -3631.679,E2 -3631.679} C_VEL
LIN {X 0,Y 545.06,Z 138.085,A -85,B 0,C 180,E1 -3634.565,E2 -3634.565} C_VEL
LIN {X 0,Y 545.03,Z 138.092,A -85,B 0,C 180,E1 -3637.305,E2 -3637.305} C_VEL
LIN {X 0,Y 545.066,Z 138.086,A -85,B 0,C 180,E1 -3640.143,E2 -3640.143} C_VEL
LIN {X 0,Y 545.044,Z 138.09,A -85,B 0,C 180,E1 -3643.11,E2 -3643.11} C_VEL
LIN {X 0,Y 545.045,Z 138.087,A -85,B 0,C 180,E1 -3646.227,E2 -3646.227} C_VEL
LIN {X 0,Y 545.071,Z 138.086,A -85,B 0,C 180,E1 -3648.885,E2 -3648.885} C_VEL
LIN {X 0,Y 545.046,Z 138.088,A -85,B 0,C 180,E1 -3651.865,E2 -3651.865} C_VEL
LIN {X 0,Y 545.035,Z 138.089,A -85,B 0,C 180,E1 -3654.532,E2 -3654.532} C_VEL
LIN {X 0,Y 545.062,Z 138.092,A -85,B 0,C 180,E1 -3657.211,E2 -3657.211} C_VEL
LIN {X 0,Y 545.062,Z 138.086,A -85,B 0,C 180,E1 -3659.811,E2 -3659.811} C_VEL
LIN {X 0,Y 545.038,Z 138.097,A -85,B 0,C 180,E1 -3662.839,E2 -3662.839} C_VEL
LIN {X 0,Y 545.021,Z 138.094,A -85,B 0,C 180,E1 -3665.63,E2 -3665.63} C_VEL
LIN {X 0,Y 545.069,Z 138.231,A -85,B 0,C 180,E1 -3666.642,E2 -3666.642} C_VEL
LIN {X 0,Y 546.101,Z 144.546,A -85,B 0,C 180,E1 -3667.691,E2 -3667.691} C_VEL
LIN {X 0,Y 545.824,Z 160.282,A -85,B 0,C 180,E1 -3670.161,E2 -3670.161} C_VEL
LIN {X 0,Y 545.507,Z 177.107,A -85,B 0,C 180,E1 -3672.763,E2 -3672.763} C_VEL
LIN {X 0,Y 545.325,Z 194.714,A -85,B 0,C 180,E1 -3675.445,E2 -3675.445} C_VEL
LIN {X 0,Y 546.509,Z 203.79,A -85,B 0,C 180,E1 -3675.597,E2 -3675.597} C_VEL
LIN {X 0,Y 546.226,Z 302.625,A -85,B 0,C 180,E1 -3676.917,E2 -3676.917} C_VEL
LIN {X 0,Y 546.052,Z 315.906,A -85,B 0,C 180,E1 -3677.243,E2 -3677.243} C_VEL
LIN {X 0,Y 545.849,Z 329.197,A -85,B 0,C 180,E1 -3677.735,E2 -3677.735} C_VEL
LIN {X 0,Y 545.652,Z 341.765,A -85,B 0,C 180,E1 -3678.38,E2 -3678.38} C_VEL
LIN {X 0,Y 545.452,Z 353.244,A -85,B 0,C 180,E1 -3679.138,E2 -3679.138} C_VEL
LIN {X 0,Y 545.234,Z 363.435,A -85,B 0,C 180,E1 -3679.979,E2 -3679.979} C_VEL
LIN {X 0,Y 545.054,Z 372.605,A -85,B 0,C 180,E1 -3680.912,E2 -3680.912} C_VEL
LIN {X 0,Y 544.892,Z 381.54,A -85,B 0,C 180,E1 -3682.03,E2 -3682.03} C_VEL
LIN {X 0,Y 544.767,Z 388.729,A -85,B 0,C 180,E1 -3683.146,E2 -3683.146} C_VEL
LIN {X 0,Y 544.741,Z 395.277,A -85,B 0,C 180,E1 -3684.447,E2 -3684.447} C_VEL
LIN {X 0,Y 544.658,Z 399.607,A -85,B 0,C 180,E1 -3685.56,E2 -3685.56} C_VEL
LIN {X 0,Y 544.669,Z 401.9,A -85,B 0,C 180,E1 -3686.301,E2 -3686.301} C_VEL
LIN {X 0,Y 544.65,Z 403.758,A -85,B 0,C 180,E1 -3687.041,E2 -3687.041} C_VEL
LIN {X 0,Y 544.546,Z 406.143,A -85,B 0,C 180,E1 -3688.521,E2 -3688.521} C_VEL
LIN {X 0,Y 544.541,Z 406.966,A -85,B 0,C 180,E1 -3690,E2 -3690} C_VEL
LIN {X 0,Y 544.546,Z 406.144,A -85,B 0,C 180,E1 -3691.479,E2 -3691.479} C_VEL
LIN {X 0,Y 544.65,Z 403.761,A -85,B 0,C 180,E1 -3692.959,E2 -3692.959} C_VEL
LIN {X 0,Y 544.684,Z 400.832,A -85,B 0,C 180,E1 -3694.069,E2 -3694.069} C_VEL
LIN {X 0,Y 544.653,Z 396.865,A -85,B 0,C 180,E1 -3695.182,E2 -3695.182} C_VEL
LIN {X 0,Y 544.714,Z 391.596,A -85,B 0,C 180,E1 -3696.328,E2 -3696.328} C_VEL
LIN {X 0,Y 544.836,Z 385.333,A -85,B 0,C 180,E1 -3697.411,E2 -3697.411} C_VEL
LIN {X 0,Y 544.988,Z 377.313,A -85,B 0,C 180,E1 -3698.528,E2 -3698.528} C_VEL
LIN {X 0,Y 545.142,Z 369.14,A -85,B 0,C 180,E1 -3699.461,E2 -3699.461} C_VEL
LIN {X 0,Y 545.365,Z 359.174,A -85,B 0,C 180,E1 -3700.394,E2 -3700.394} C_VEL
LIN {X 0,Y 545.569,Z 348.34,A -85,B 0,C 180,E1 -3701.208,E2 -3701.208} C_VEL
LIN {X 0,Y 545.712,Z 336.891,A -85,B 0,C 180,E1 -3701.891,E2 -3701.891} C_VEL
LIN {X 0,Y 545.938,Z 324.671,A -85,B 0,C 180,E1 -3702.452,E2 -3702.452} C_VEL
LIN {X 0,Y 546.092,Z 311.856,A -85,B 0,C 180,E1 -3702.874,E2 -3702.874} C_VEL
LIN {X 0,Y 546.271,Z 298.272,A -85,B 0,C 180,E1 -3703.153,E2 -3703.153} C_VEL
LIN {X 0,Y 546.444,Z 202.115,A -85,B 0,C 180,E1 -3704.427,E2 -3704.427} C_VEL
LIN {X 0,Y 545.318,Z 194.473,A -85,B 0,C 180,E1 -3704.579,E2 -3704.579} C_VEL
LIN {X 0,Y 545.571,Z 174.829,A -85,B 0,C 180,E1 -3707.586,E2 -3707.586} C_VEL
LIN {X 0,Y 545.929,Z 154.556,A -85,B 0,C 180,E1 -3710.733,E2 -3710.733} C_VEL
LIN {X 0,Y 546.096,Z 144.319,A -85,B 0,C 180,E1 -3712.345,E2 -3712.345} C_VEL
LIN {X 0,Y 545.075,Z 138.092,A -85,B 0,C 180,E1 -3713.408,E2 -3713.408} C_VEL
LIN {X 0,Y 545.049,Z 138.088,A -85,B 0,C 180,E1 -3716.002,E2 -3716.002} C_VEL
LIN {X 0,Y 545.045,Z 138.091,A -85,B 0,C 180,E1 -3718.739,E2 -3718.739} C_VEL
LIN {X 0,Y 545.045,Z 138.087,A -85,B 0,C 180,E1 -3721.676,E2 -3721.676} C_VEL
LIN {X 0,Y 545.058,Z 138.089,A -85,B 0,C 180,E1 -3724.565,E2 -3724.565} C_VEL
LIN {X 0,Y 545.035,Z 138.09,A -85,B 0,C 180,E1 -3727.304,E2 -3727.304} C_VEL
LIN {X 0,Y 545.063,Z 138.086,A -85,B 0,C 180,E1 -3730.143,E2 -3730.143} C_VEL
LIN {X 0,Y 545.039,Z 138.096,A -85,B 0,C 180,E1 -3732.694,E2 -3732.694} C_VEL
LIN {X 0,Y 545.029,Z 138.09,A -85,B 0,C 180,E1 -3735.17,E2 -3735.17} C_VEL
LIN {X 0,Y 545.061,Z 138.086,A -85,B 0,C 180,E1 -3737.895,E2 -3737.895} C_VEL
LIN {X 0,Y 545.08,Z 138.085,A -85,B 0,C 180,E1 -3740.818,E2 -3740.818} C_VEL
LIN {X 0,Y 545.034,Z 138.089,A -85,B 0,C 180,E1 -3743.619,E2 -3743.619} C_VEL
LIN {X 0,Y 545.065,Z 138.092,A -85,B 0,C 180,E1 -3746.328,E2 -3746.328} C_VEL
LIN {X 0,Y 545.063,Z 138.085,A -85,B 0,C 180,E1 -3748.952,E2 -3748.952} C_VEL
LIN {X 0,Y 545.08,Z 138.084,A -85,B 0,C 180,E1 -3751.506,E2 -3751.506} C_VEL
LIN {X 0,Y 545.082,Z 138.084,A -85,B 0,C 180,E1 -3754.494,E2 -3754.494} C_VEL
LIN {X 0,Y 545.036,Z 138.089,A -85,B 0,C 180,E1 -3757.242,E2 -3757.242} C_VEL
LIN {X 0,Y 545.116,Z 138.079,A -85,B 0,C 180,E1 -3760.415,E2 -3760.415} C_VEL
LIN {X 0,Y 545.063,Z 138.091,A -85,B 0,C 180,E1 -3763.521,E2 -3763.521} C_VEL
LIN {X 0,Y 545.094,Z 138.087,A -85,B 0,C 180,E1 -3765.82,E2 -3765.82} C_VEL
LIN {X 0,Y 545.118,Z 138.078,A -85,B 0,C 180,E1 -3768.849,E2 -3768.849} C_VEL
LIN {X 0,Y 545.125,Z 138.08,A -85,B 0,C 180,E1 -3771.847,E2 -3771.847} C_VEL
LIN {X 0,Y 545.205,Z 138.068,A -85,B 0,C 180,E1 -3774.823,E2 -3774.823} C_VEL
LIN {X 0,Y 545.199,Z 138.07,A -85,B 0,C 180,E1 -3777.784,E2 -3777.784} C_VEL
LIN {X 0,Y 545.209,Z 138.069,A -85,B 0,C 180,E1 -3780.739,E2 -3780.739} C_VEL
LIN {X 0,Y 545.169,Z 138.078,A -85,B 0,C 180,E1 -3782.956,E2 -3782.956} C_VEL
LIN {X 0,Y 545.171,Z 138.071,A -85,B 0,C 180,E1 -3785.92,E2 -3785.92} C_VEL
LIN {X 0,Y 545.111,Z 138.087,A -85,B 0,C 180,E1 -3788.9,E2 -3788.9} C_VEL
LIN {X 0,Y 545.135,Z 138.075,A -85,B 0,C 180,E1 -3791.904,E2 -3791.904} C_VEL
LIN {X 0,Y 545.086,Z 138.088,A -85,B 0,C 180,E1 -3794.944,E2 -3794.944} C_VEL
LIN {X 0,Y 545.079,Z 138.083,A -85,B 0,C 180,E1 -3798.026,E2 -3798.026} C_VEL
LIN {X 0,Y 545.096,Z 138.086,A -85,B 0,C 180,E1 -3800.372,E2 -3800.372} C_VEL
LIN {X 0,Y 545.081,Z 138.082,A -85,B 0,C 180,E1 -3803.559,E2 -3803.559} C_VEL
LIN {X 0,Y 545.081,Z 138.085,A -85,B 0,C 180,E1 -3806.001,E2 -3806.001} C_VEL
LIN {X 0,Y 545.09,Z 138.085,A -85,B 0,C 180,E1 -3808.748,E2 -3808.748} C_VEL
LIN {X 0,Y 545.058,Z 138.086,A -85,B 0,C 180,E1 -3811.679,E2 -3811.679} C_VEL
LIN {X 0,Y 545.063,Z 138.088,A -85,B 0,C 180,E1 -3814.565,E2 -3814.565} C_VEL
LIN {X 0,Y 545.063,Z 138.084,A -85,B 0,C 180,E1 -3816.994,E2 -3816.994} C_VEL
LIN {X 0,Y 544.357,Z 138.176,A -85,B 0,C 180,E1 -3817.61,E2 -3817.61} C_VEL
LIN {X 0,Y 541.494,Z 138.531,A -85,B 0,C 180,E1 -3818.611,E2 -3818.611} C_VEL
LIN {X 0,Y 539.108,Z 138.829,A -85,B 0,C 180,E1 -3819.417,E2 -3819.417} C_VEL
LIN {X 0,Y 538.098,Z 138.962,A -85,B 0,C 180,E1 -3820.039,E2 -3820.039} C_VEL
LIN {X 0,Y 538.022,Z 138.962,A -85,B 0,C 180,E1 -3820.25,E2 -3820.25} C_VEL
LIN {X 0,Y 538.027,Z 138.961,A -85,B 0,C 180,E1 -3822.988,E2 -3822.988} C_VEL
LIN {X 0,Y 538.031,Z 138.969,A -85,B 0,C 180,E1 -3825.926,E2 -3825.926} C_VEL
LIN {X 0,Y 538.05,Z 138.96,A -85,B 0,C 180,E1 -3829.253,E2 -3829.253} C_VEL
LIN {X 0,Y 537.994,Z 138.968,A -85,B 0,C 180,E1 -3832.123,E2 -3832.123} C_VEL
LIN {X 0,Y 537.999,Z 138.965,A -85,B 0,C 180,E1 -3834.916,E2 -3834.916} C_VEL
LIN {X 0,Y 538.019,Z 138.97,A -85,B 0,C 180,E1 -3837.617,E2 -3837.617} C_VEL
LIN {X 0,Y 538.017,Z 138.962,A -85,B 0,C 180,E1 -3840.239,E2 -3840.239} C_VEL
LIN {X 0,Y 538.057,Z 138.959,A -85,B 0,C 180,E1 -3842.796,E2 -3842.796} C_VEL
LIN {X 0,Y 538.05,Z 138.966,A -85,B 0,C 180,E1 -3845.293,E2 -3845.293} C_VEL
LIN {X 0,Y 538.027,Z 138.965,A -85,B 0,C 180,E1 -3848.546,E2 -3848.546} C_VEL
LIN {X 0,Y 538.063,Z 138.985,A -85,B 0,C 180,E1 -3849.395,E2 -3849.395} C_VEL
LIN {X 0,Y 538.631,Z 143.062,A -85,B 0,C 180,E1 -3850.169,E2 -3850.169} C_VEL
LIN {X 0,Y 538.451,Z 156.034,A -85,B 0,C 180,E1 -3852.53,E2 -3852.53} C_VEL
LIN {X 0,Y 538.274,Z 171.714,A -85,B 0,C 180,E1 -3855.308,E2 -3855.308} C_VEL
LIN {X 0,Y 539.736,Z 179.959,A -85,B 0,C 180,E1 -3855.46,E2 -3855.46} C_VEL
LIN {X 0,Y 539.322,Z 278.614,A -85,B 0,C 180,E1 -3856.794,E2 -3856.794} C_VEL
LIN {X 0,Y 539.171,Z 291.816,A -85,B 0,C 180,E1 -3857.126,E2 -3857.126} C_VEL
LIN {X 0,Y 538.971,Z 303.928,A -85,B 0,C 180,E1 -3857.575,E2 -3857.575} C_VEL
LIN {X 0,Y 538.826,Z 315.021,A -85,B 0,C 180,E1 -3858.128,E2 -3858.128} C_VEL
LIN {X 0,Y 538.589,Z 325.75,A -85,B 0,C 180,E1 -3858.808,E2 -3858.808} C_VEL
LIN {X 0,Y 538.338,Z 336.457,A -85,B 0,C 180,E1 -3859.659,E2 -3859.659} C_VEL
LIN {X 0,Y 538.146,Z 346.089,A -85,B 0,C 180,E1 -3860.605,E2 -3860.605} C_VEL
LIN {X 0,Y 537.955,Z 353.98,A -85,B 0,C 180,E1 -3861.548,E2 -3861.548} C_VEL
LIN {X 0,Y 537.771,Z 361.699,A -85,B 0,C 180,E1 -3862.679,E2 -3862.679} C_VEL
LIN {X 0,Y 537.729,Z 368.773,A -85,B 0,C 180,E1 -3863.998,E2 -3863.998} C_VEL
LIN {X 0,Y 537.545,Z 373.494,A -85,B 0,C 180,E1 -3865.125,E2 -3865.125} C_VEL
LIN {X 0,Y 537.591,Z 377.106,A -85,B 0,C 180,E1 -3866.252,E2 -3866.252} C_VEL
LIN {X 0,Y 537.58,Z 378.974,A -85,B 0,C 180,E1 -3867.002,E2 -3867.002} C_VEL
LIN {X 0,Y 537.49,Z 380.387,A -85,B 0,C 180,E1 -3867.752,E2 -3867.752} C_VEL
LIN {X 0,Y 537.445,Z 382.008,A -85,B 0,C 180,E1 -3869.251,E2 -3869.251} C_VEL
LIN {X 0,Y 537.445,Z 382.247,A -85,B 0,C 180,E1 -3870,E2 -3870} C_VEL
LIN {X 0,Y 537.445,Z 382.065,A -85,B 0,C 180,E1 -3870.749,E2 -3870.749} C_VEL
LIN {X 0,Y 537.49,Z 380.518,A -85,B 0,C 180,E1 -3872.248,E2 -3872.248} C_VEL
LIN {X 0,Y 537.58,Z 379.162,A -85,B 0,C 180,E1 -3872.998,E2 -3872.998} C_VEL
LIN {X 0,Y 537.604,Z 376.299,A -85,B 0,C 180,E1 -3874.123,E2 -3874.123} C_VEL
LIN {X 0,Y 537.587,Z 372.417,A -85,B 0,C 180,E1 -3875.251,E2 -3875.251} C_VEL
LIN {X 0,Y 537.683,Z 367.584,A -85,B 0,C 180,E1 -3876.341,E2 -3876.341} C_VEL
LIN {X 0,Y 537.809,Z 361.101,A -85,B 0,C 180,E1 -3877.509,E2 -3877.509} C_VEL
LIN {X 0,Y 537.971,Z 353.205,A -85,B 0,C 180,E1 -3878.64,E2 -3878.64} C_VEL
LIN {X 0,Y 538.177,Z 343.382,A -85,B 0,C 180,E1 -3879.774,E2 -3879.774} C_VEL
LIN {X 0,Y 538.442,Z 333.084,A -85,B 0,C 180,E1 -3880.719,E2 -3880.719} C_VEL
LIN {X 0,Y 538.662,Z 321.882,A -85,B 0,C 180,E1 -3881.544,E2 -3881.544} C_VEL
LIN {X 0,Y 538.923,Z 309.915,A -85,B 0,C 180,E1 -3882.234,E2 -3882.234} C_VEL
LIN {X 0,Y 539.112,Z 297.908,A -85,B 0,C 180,E1 -3882.756,E2 -3882.756} C_VEL
LIN {X 0,Y 539.251,Z 284.852,A -85,B 0,C 180,E1 -3883.16,E2 -3883.16} C_VEL
LIN {X 0,Y 539.419,Z 272.415,A -85,B 0,C 180,E1 -3883.395,E2 -3883.395} C_VEL
LIN {X 0,Y 539.604,Z 179.147,A -85,B 0,C 180,E1 -3884.644,E2 -3884.644} C_VEL
LIN {X 0,Y 538.242,Z 171.467,A -85,B 0,C 180,E1 -3884.797,E2 -3884.797} C_VEL
LIN {X 0,Y 538.529,Z 154.14,A -85,B 0,C 180,E1 -3887.9,E2 -3887.9} C_VEL
LIN {X 0,Y 538.609,Z 142.455,A -85,B 0,C 180,E1 -3890.034,E2 -3890.034} C_VEL
LIN {X 0,Y 538.046,Z 138.968,A -85,B 0,C 180,E1 -3890.701,E2 -3890.701} C_VEL
LIN {X 0,Y 538.002,Z 138.965,A -85,B 0,C 180,E1 -3893.888,E2 -3893.888} C_VEL
LIN {X 0,Y 538.043,Z 138.963,A -85,B 0,C 180,E1 -3896.366,E2 -3896.366} C_VEL
LIN {X 0,Y 538.032,Z 138.966,A -85,B 0,C 180,E1 -3898.933,E2 -3898.933} C_VEL
LIN {X 0,Y 538.011,Z 138.964,A -85,B 0,C 180,E1 -3901.887,E2 -3901.887} C_VEL
LIN {X 0,Y 538.011,Z 138.97,A -85,B 0,C 180,E1 -3904.617,E2 -3904.617} C_VEL
LIN {X 0,Y 538.005,Z 138.964,A -85,B 0,C 180,E1 -3907.17,E2 -3907.17} C_VEL
LIN {X 0,Y 538.024,Z 138.963,A -85,B 0,C 180,E1 -3909.797,E2 -3909.797} C_VEL
LIN {X 0,Y 538.02,Z 138.964,A -85,B 0,C 180,E1 -3912.786,E2 -3912.786} C_VEL
LIN {X 0,Y 538.033,Z 138.96,A -85,B 0,C 180,E1 -3915.14,E2 -3915.14} C_VEL
LIN {X 0,Y 538.035,Z 138.967,A -85,B 0,C 180,E1 -3918.227,E2 -3918.227} C_VEL
LIN {X 0,Y 538.016,Z 138.963,A -85,B 0,C 180,E1 -3921.17,E2 -3921.17} C_VEL
LIN {X 0,Y 537.994,Z 138.971,A -85,B 0,C 180,E1 -3924.088,E2 -3924.088} C_VEL
LIN {X 0,Y 538.03,Z 138.961,A -85,B 0,C 180,E1 -3926.727,E2 -3926.727} C_VEL
LIN {X 0,Y 538.026,Z 138.967,A -85,B 0,C 180,E1 -3929.556,E2 -3929.556} C_VEL
LIN {X 0,Y 538.04,Z 138.964,A -85,B 0,C 180,E1 -3931.95,E2 -3931.95} C_VEL
LIN {X 0,Y 538.071,Z 138.955,A -85,B 0,C 180,E1 -3934.467,E2 -3934.467} C_VEL
LIN {X 0,Y 537.993,Z 138.971,A -85,B 0,C 180,E1 -3937.738,E2 -3937.738} C_VEL
LIN {X 0,Y 538.079,Z 138.955,A -85,B 0,C 180,E1 -3940.148,E2 -3940.148} C_VEL
LIN {X 0,Y 538.025,Z 138.97,A -85,B 0,C 180,E1 -3943.299,E2 -3943.299} C_VEL
LIN {X 0,Y 538.063,Z 138.96,A -85,B 0,C 180,E1 -3945.631,E2 -3945.631} C_VEL
LIN {X 0,Y 538.077,Z 138.957,A -85,B 0,C 180,E1 -3948.701,E2 -3948.701} C_VEL
LIN {X 0,Y 538.085,Z 138.955,A -85,B 0,C 180,E1 -3951.74,E2 -3951.74} C_VEL
LIN {X 0,Y 538.161,Z 138.95,A -85,B 0,C 180,E1 -3954.755,E2 -3954.755} C_VEL
LIN {X 0,Y 538.169,Z 138.943,A -85,B 0,C 180,E1 -3957.755,E2 -3957.755} C_VEL
LIN {X 0,Y 538.184,Z 138.95,A -85,B 0,C 180,E1 -3960.748,E2 -3960.748} C_VEL
LIN {X 0,Y 538.136,Z 138.952,A -85,B 0,C 180,E1 -3962.994,E2 -3962.994} C_VEL
LIN {X 0,Y 538.121,Z 138.95,A -85,B 0,C 180,E1 -3965.997,E2 -3965.997} C_VEL
LIN {X 0,Y 538.061,Z 138.959,A -85,B 0,C 180,E1 -3969.018,E2 -3969.018} C_VEL
LIN {X 0,Y 538.082,Z 138.958,A -85,B 0,C 180,E1 -3972.063,E2 -3972.063} C_VEL
LIN {X 0,Y 538.044,Z 138.959,A -85,B 0,C 180,E1 -3975.144,E2 -3975.144} C_VEL
LIN {X 0,Y 538.024,Z 138.971,A -85,B 0,C 180,E1 -3978.271,E2 -3978.271} C_VEL
LIN {X 0,Y 538.036,Z 138.962,A -85,B 0,C 180,E1 -3980.652,E2 -3980.652} C_VEL
LIN {X 0,Y 538.002,Z 138.97,A -85,B 0,C 180,E1 -3983.889,E2 -3983.889} C_VEL
LIN {X 0,Y 538.036,Z 138.964,A -85,B 0,C 180,E1 -3986.367,E2 -3986.367} C_VEL
LIN {X 0,Y 538.029,Z 138.961,A -85,B 0,C 180,E1 -3988.933,E2 -3988.933} C_VEL
LIN {X 0,Y 538.009,Z 138.972,A -85,B 0,C 180,E1 -3991.887,E2 -3991.887} C_VEL
LIN {X 0,Y 538.01,Z 138.963,A -85,B 0,C 180,E1 -3994.618,E2 -3994.618} C_VEL
LIN {X 0,Y 537.999,Z 138.967,A -85,B 0,C 180,E1 -3997.169,E2 -3997.169} C_VEL
LIN {X 0,Y 538.023,Z 138.968,A -85,B 0,C 180,E1 -3999.797,E2 -3999.797} C_VEL
LIN {X 0,Y 537.999,Z 138.965,A -85,B 0,C 180,E1 -4002.788,E2 -4002.788} C_VEL
LIN {X 0,Y 537.997,Z 138.969,A -85,B 0,C 180,E1 -4005.137,E2 -4005.137} C_VEL
LIN {X 0,Y 538.018,Z 138.962,A -85,B 0,C 180,E1 -4008.226,E2 -4008.226} C_VEL
LIN {X 0,Y 538.01,Z 138.971,A -85,B 0,C 180,E1 -4011.169,E2 -4011.169} C_VEL
LIN {X 0,Y 537.994,Z 138.965,A -85,B 0,C 180,E1 -4014.089,E2 -4014.089} C_VEL
LIN {X 0,Y 538.032,Z 138.964,A -85,B 0,C 180,E1 -4016.728,E2 -4016.728} C_VEL
LIN {X 0,Y 538.002,Z 138.968,A -85,B 0,C 180,E1 -4019.561,E2 -4019.561} C_VEL
LIN {X 0,Y 538.008,Z 138.969,A -85,B 0,C 180,E1 -4022.659,E2 -4022.659} C_VEL
LIN {X 0,Y 537.983,Z 138.974,A -85,B 0,C 180,E1 -4025.29,E2 -4025.29} C_VEL
LIN {X 0,Y 538.039,Z 139.031,A -85,B 0,C 180,E1 -4026.472,E2 -4026.472} C_VEL
LIN {X 0,Y 539.085,Z 144.628,A -85,B 0,C 180,E1 -4027.422,E2 -4027.422} C_VEL
LIN {X 0,Y 538.881,Z 158.904,A -85,B 0,C 180,E1 -4029.699,E2 -4029.699} C_VEL
LIN {X 0,Y 538.542,Z 176.948,A -85,B 0,C 180,E1 -4032.533,E2 -4032.533} C_VEL
LIN {X 0,Y 538.291,Z 194.381,A -85,B 0,C 180,E1 -4035.238,E2 -4035.238} C_VEL
LIN {X 0,Y 539.638,Z 203.857,A -85,B 0,C 180,E1 -4035.413,E2 -4035.413} C_VEL
LIN {X 0,Y 539.316,Z 302.463,A -85,B 0,C 180,E1 -4036.746,E2 -4036.746} C_VEL
LIN {X 0,Y 539.139,Z 315.745,A -85,B 0,C 180,E1 -4037.077,E2 -4037.077} C_VEL
LIN {X 0,Y 538.903,Z 329.035,A -85,B 0,C 180,E1 -4037.574,E2 -4037.574} C_VEL
LIN {X 0,Y 538.685,Z 339.805,A -85,B 0,C 180,E1 -4038.119,E2 -4038.119} C_VEL
LIN {X 0,Y 538.466,Z 351.787,A -85,B 0,C 180,E1 -4038.9,E2 -4038.9} C_VEL
LIN {X 0,Y 538.236,Z 362.228,A -85,B 0,C 180,E1 -4039.752,E2 -4039.752} C_VEL
LIN {X 0,Y 538.062,Z 370.764,A -85,B 0,C 180,E1 -4040.603,E2 -4040.603} C_VEL
LIN {X 0,Y 537.899,Z 378.64,A -85,B 0,C 180,E1 -4041.548,E2 -4041.548} C_VEL
LIN {X 0,Y 537.754,Z 386.331,A -85,B 0,C 180,E1 -4042.679,E2 -4042.679} C_VEL
LIN {X 0,Y 537.693,Z 393.421,A -85,B 0,C 180,E1 -4043.998,E2 -4043.998} C_VEL
LIN {X 0,Y 537.54,Z 398.134,A -85,B 0,C 180,E1 -4045.125,E2 -4045.125} C_VEL
LIN {X 0,Y 537.591,Z 401.738,A -85,B 0,C 180,E1 -4046.252,E2 -4046.252} C_VEL
LIN {X 0,Y 537.551,Z 403.595,A -85,B 0,C 180,E1 -4047.002,E2 -4047.002} C_VEL
LIN {X 0,Y 537.451,Z 405.981,A -85,B 0,C 180,E1 -4048.501,E2 -4048.501} C_VEL
LIN {X 0,Y 537.444,Z 406.804,A -85,B 0,C 180,E1 -4050,E2 -4050} C_VEL
LIN {X 0,Y 537.451,Z 405.982,A -85,B 0,C 180,E1 -4051.499,E2 -4051.499} C_VEL
LIN {X 0,Y 537.551,Z 403.599,A -85,B 0,C 180,E1 -4052.998,E2 -4052.998} C_VEL
LIN {X 0,Y 537.603,Z 400.67,A -85,B 0,C 180,E1 -4054.123,E2 -4054.123} C_VEL
LIN {X 0,Y 537.587,Z 396.703,A -85,B 0,C 180,E1 -4055.251,E2 -4055.251} C_VEL
LIN {X 0,Y 537.621,Z 391.929,A -85,B 0,C 180,E1 -4056.312,E2 -4056.312} C_VEL
LIN {X 0,Y 537.757,Z 385.17,A -85,B 0,C 180,E1 -4057.51,E2 -4057.51} C_VEL
LIN {X 0,Y 537.918,Z 377.15,A -85,B 0,C 180,E1 -4058.641,E2 -4058.641} C_VEL
LIN {X 0,Y 538.112,Z 368.978,A -85,B 0,C 180,E1 -4059.586,E2 -4059.586} C_VEL
LIN {X 0,Y 538.347,Z 359.011,A -85,B 0,C 180,E1 -4060.531,E2 -4060.531} C_VEL
LIN {X 0,Y 538.557,Z 349.18,A -85,B 0,C 180,E1 -4061.288,E2 -4061.288} C_VEL
LIN {X 0,Y 538.721,Z 338.129,A -85,B 0,C 180,E1 -4061.972,E2 -4061.972} C_VEL
LIN {X 0,Y 538.982,Z 325.64,A -85,B 0,C 180,E1 -4062.568,E2 -4062.568} C_VEL
LIN {X 0,Y 539.143,Z 312.607,A -85,B 0,C 180,E1 -4063.019,E2 -4063.019} C_VEL
LIN {X 0,Y 539.362,Z 299.615,A -85,B 0,C 180,E1 -4063.301,E2 -4063.301} C_VEL
LIN {X 0,Y 539.533,Z 202.515,A -85,B 0,C 180,E1 -4064.608,E2 -4064.608} C_VEL
LIN {X 0,Y 538.287,Z 194.363,A -85,B 0,C 180,E1 -4064.765,E2 -4064.765} C_VEL
LIN {X 0,Y 538.58,Z 175.364,A -85,B 0,C 180,E1 -4067.713,E2 -4067.713} C_VEL
LIN {X 0,Y 538.971,Z 155.659,A -85,B 0,C 180,E1 -4070.814,E2 -4070.814} C_VEL
LIN {X 0,Y 539.166,Z 145.76,A -85,B 0,C 180,E1 -4072.392,E2 -4072.392} C_VEL
LIN {X 0,Y 538.049,Z 138.967,A -85,B 0,C 180,E1 -4073.577,E2 -4073.577} C_VEL
LIN {X 0,Y 538.012,Z 138.965,A -85,B 0,C 180,E1 -4076.368,E2 -4076.368} C_VEL
LIN {X 0,Y 537.993,Z 138.971,A -85,B 0,C 180,E1 -4078.926,E2 -4078.926} C_VEL
LIN {X 0,Y 538,Z 138.964,A -85,B 0,C 180,E1 -4081.885,E2 -4081.885} C_VEL
LIN {X 0,Y 538.008,Z 138.968,A -85,B 0,C 180,E1 -4084.617,E2 -4084.617} C_VEL
LIN {X 0,Y 538.004,Z 138.968,A -85,B 0,C 180,E1 -4087.169,E2 -4087.169} C_VEL
LIN {X 0,Y 538.008,Z 138.963,A -85,B 0,C 180,E1 -4089.798,E2 -4089.798} C_VEL
LIN {X 0,Y 537.988,Z 138.973,A -85,B 0,C 180,E1 -4092.789,E2 -4092.789} C_VEL
LIN {X 0,Y 538,Z 138.966,A -85,B 0,C 180,E1 -4095.137,E2 -4095.137} C_VEL
LIN {X 0,Y 538.019,Z 138.967,A -85,B 0,C 180,E1 -4098.225,E2 -4098.225} C_VEL
LIN {X 0,Y 538.012,Z 138.963,A -85,B 0,C 180,E1 -4101.169,E2 -4101.169} C_VEL
LIN {X 0,Y 537.989,Z 138.972,A -85,B 0,C 180,E1 -4104.089,E2 -4104.089} C_VEL
LIN {X 0,Y 538.03,Z 138.963,A -85,B 0,C 180,E1 -4106.727,E2 -4106.727} C_VEL
LIN {X 0,Y 538.011,Z 138.964,A -85,B 0,C 180,E1 -4109.559,E2 -4109.559} C_VEL
LIN {X 0,Y 538.019,Z 138.969,A -85,B 0,C 180,E1 -4111.949,E2 -4111.949} C_VEL
LIN {X 0,Y 538.059,Z 138.96,A -85,B 0,C 180,E1 -4114.466,E2 -4114.466} C_VEL
LIN {X 0,Y 538.013,Z 138.963,A -85,B 0,C 180,E1 -4116.928,E2 -4116.928} C_VEL
LIN {X 0,Y 538.08,Z 138.959,A -85,B 0,C 180,E1 -4120.148,E2 -4120.148} C_VEL
LIN {X 0,Y 538.011,Z 138.966,A -85,B 0,C 180,E1 -4123.299,E2 -4123.299} C_VEL
LIN {X 0,Y 538.063,Z 138.965,A -85,B 0,C 180,E1 -4125.631,E2 -4125.631} C_VEL
LIN {X 0,Y 538.077,Z 138.955,A -85,B 0,C 180,E1 -4128.702,E2 -4128.702} C_VEL
LIN {X 0,Y 538.082,Z 138.959,A -85,B 0,C 180,E1 -4131.74,E2 -4131.74} C_VEL
LIN {X 0,Y 538.162,Z 138.945,A -85,B 0,C 180,E1 -4134.755,E2 -4134.755} C_VEL
LIN {X 0,Y 538.17,Z 138.946,A -85,B 0,C 180,E1 -4137.755,E2 -4137.755} C_VEL
LIN {X 0,Y 538.18,Z 138.945,A -85,B 0,C 180,E1 -4140.748,E2 -4140.748} C_VEL
LIN {X 0,Y 538.136,Z 138.954,A -85,B 0,C 180,E1 -4142.995,E2 -4142.995} C_VEL
LIN {X 0,Y 538.12,Z 138.949,A -85,B 0,C 180,E1 -4145.997,E2 -4145.997} C_VEL
LIN {X 0,Y 538.061,Z 138.965,A -85,B 0,C 180,E1 -4149.018,E2 -4149.018} C_VEL
LIN {X 0,Y 538.083,Z 138.954,A -85,B 0,C 180,E1 -4152.063,E2 -4152.063} C_VEL
LIN {X 0,Y 538.045,Z 138.962,A -85,B 0,C 180,E1 -4155.144,E2 -4155.144} C_VEL
LIN {X 0,Y 538.032,Z 138.964,A -85,B 0,C 180,E1 -4158.27,E2 -4158.27} C_VEL
LIN {X 0,Y 538.04,Z 138.968,A -85,B 0,C 180,E1 -4160.651,E2 -4160.651} C_VEL
LIN {X 0,Y 538.004,Z 138.965,A -85,B 0,C 180,E1 -4163.888,E2 -4163.888} C_VEL
LIN {X 0,Y 538.043,Z 138.967,A -85,B 0,C 180,E1 -4166.367,E2 -4166.367} C_VEL
LIN {X 0,Y 538.031,Z 138.962,A -85,B 0,C 180,E1 -4168.934,E2 -4168.934} C_VEL
LIN {X 0,Y 538.011,Z 138.966,A -85,B 0,C 180,E1 -4171.887,E2 -4171.887} C_VEL
LIN {X 0,Y 538.012,Z 138.966,A -85,B 0,C 180,E1 -4174.618,E2 -4174.618} C_VEL
LIN {X 0,Y 538.005,Z 138.964,A -85,B 0,C 180,E1 -4177.17,E2 -4177.17} C_VEL
LIN {X 0,Y 538.022,Z 138.962,A -85,B 0,C 180,E1 -4180.25,E2 -4180.25} C_VEL
LIN {X 0,Y 537.371,Z 139.044,A -85,B 0,C 180,E1 -4180.875,E2 -4180.875} C_VEL
LIN {X 0,Y 534.523,Z 139.405,A -85,B 0,C 180,E1 -4181.89,E2 -4181.89} C_VEL
LIN {X 0,Y 532.1,Z 139.707,A -85,B 0,C 180,E1 -4182.707,E2 -4182.707} C_VEL
LIN {X 0,Y 531.052,Z 139.834,A -85,B 0,C 180,E1 -4183.338,E2 -4183.338} C_VEL
LIN {X 0,Y 530.964,Z 139.843,A -85,B 0,C 180,E1 -4183.552,E2 -4183.552} C_VEL
LIN {X 0,Y 530.966,Z 139.841,A -85,B 0,C 180,E1 -4186.506,E2 -4186.506} C_VEL
LIN {X 0,Y 530.983,Z 139.845,A -85,B 0,C 180,E1 -4189.567,E2 -4189.567} C_VEL
LIN {X 0,Y 530.969,Z 139.84,A -85,B 0,C 180,E1 -4192.577,E2 -4192.577} C_VEL
LIN {X 0,Y 530.982,Z 139.844,A -85,B 0,C 180,E1 -4195.31,E2 -4195.31} C_VEL
LIN {X 0,Y 530.968,Z 139.842,A -85,B 0,C 180,E1 -4198.032,E2 -4198.032} C_VEL
LIN {X 0,Y 530.99,Z 139.839,A -85,B 0,C 180,E1 -4200.875,E2 -4200.875} C_VEL
LIN {X 0,Y 531.003,Z 139.844,A -85,B 0,C 180,E1 -4203.256,E2 -4203.256} C_VEL
LIN {X 0,Y 530.986,Z 139.84,A -85,B 0,C 180,E1 -4205.961,E2 -4205.961} C_VEL
LIN {X 0,Y 531.022,Z 139.845,A -85,B 0,C 180,E1 -4209.266,E2 -4209.266} C_VEL
LIN {X 0,Y 531.675,Z 145.245,A -85,B 0,C 180,E1 -4210.301,E2 -4210.301} C_VEL
LIN {X 0,Y 531.452,Z 159.331,A -85,B 0,C 180,E1 -4212.888,E2 -4212.888} C_VEL
LIN {X 0,Y 531.254,Z 171.593,A -85,B 0,C 180,E1 -4215.098,E2 -4215.098} C_VEL
LIN {X 0,Y 532.86,Z 181.245,A -85,B 0,C 180,E1 -4215.283,E2 -4215.283} C_VEL
LIN {X 0,Y 532.441,Z 278.805,A -85,B 0,C 180,E1 -4216.62,E2 -4216.62} C_VEL
LIN {X 0,Y 532.273,Z 291.997,A -85,B 0,C 180,E1 -4216.956,E2 -4216.956} C_VEL
LIN {X 0,Y 532.06,Z 304.104,A -85,B 0,C 180,E1 -4217.411,E2 -4217.411} C_VEL
LIN {X 0,Y 531.883,Z 315.812,A -85,B 0,C 180,E1 -4218.006,E2 -4218.006} C_VEL
LIN {X 0,Y 531.603,Z 327.207,A -85,B 0,C 180,E1 -4218.755,E2 -4218.755} C_VEL
LIN {X 0,Y 531.317,Z 337.692,A -85,B 0,C 180,E1 -4219.617,E2 -4219.617} C_VEL
LIN {X 0,Y 531.121,Z 346.258,A -85,B 0,C 180,E1 -4220.479,E2 -4220.479} C_VEL
LIN {X 0,Y 530.924,Z 354.147,A -85,B 0,C 180,E1 -4221.436,E2 -4221.436} C_VEL
LIN {X 0,Y 530.734,Z 361.864,A -85,B 0,C 180,E1 -4222.582,E2 -4222.582} C_VEL
LIN {X 0,Y 530.661,Z 368.939,A -85,B 0,C 180,E1 -4223.918,E2 -4223.918} C_VEL
LIN {X 0,Y 530.463,Z 373.658,A -85,B 0,C 180,E1 -4225.06,E2 -4225.06} C_VEL
LIN {X 0,Y 530.517,Z 377.269,A -85,B 0,C 180,E1 -4226.202,E2 -4226.202} C_VEL
LIN {X 0,Y 530.512,Z 379.137,A -85,B 0,C 180,E1 -4226.962,E2 -4226.962} C_VEL
LIN {X 0,Y 530.413,Z 380.549,A -85,B 0,C 180,E1 -4227.722,E2 -4227.722} C_VEL
LIN {X 0,Y 530.347,Z 382.17,A -85,B 0,C 180,E1 -4229.241,E2 -4229.241} C_VEL
LIN {X 0,Y 530.347,Z 382.409,A -85,B 0,C 180,E1 -4230,E2 -4230} C_VEL
LIN {X 0,Y 530.347,Z 382.227,A -85,B 0,C 180,E1 -4230.759,E2 -4230.759} C_VEL
LIN {X 0,Y 530.413,Z 380.679,A -85,B 0,C 180,E1 -4232.278,E2 -4232.278} C_VEL
LIN {X 0,Y 530.512,Z 379.322,A -85,B 0,C 180,E1 -4233.037,E2 -4233.037} C_VEL
LIN {X 0,Y 530.525,Z 376.46,A -85,B 0,C 180,E1 -4234.178,E2 -4234.178} C_VEL
LIN {X 0,Y 530.524,Z 372.577,A -85,B 0,C 180,E1 -4235.321,E2 -4235.321} C_VEL
LIN {X 0,Y 530.616,Z 366.903,A -85,B 0,C 180,E1 -4236.597,E2 -4236.597} C_VEL
LIN {X 0,Y 530.785,Z 360.036,A -85,B 0,C 180,E1 -4237.8,E2 -4237.8} C_VEL
LIN {X 0,Y 530.959,Z 351.884,A -85,B 0,C 180,E1 -4238.947,E2 -4238.947} C_VEL
LIN {X 0,Y 531.182,Z 343.539,A -85,B 0,C 180,E1 -4239.904,E2 -4239.904} C_VEL
LIN {X 0,Y 531.456,Z 333.239,A -85,B 0,C 180,E1 -4240.862,E2 -4240.862} C_VEL
LIN {X 0,Y 531.703,Z 322.341,A -85,B 0,C 180,E1 -4241.676,E2 -4241.676} C_VEL
LIN {X 0,Y 531.94,Z 311.876,A -85,B 0,C 180,E1 -4242.301,E2 -4242.301} C_VEL
LIN {X 0,Y 532.128,Z 300.57,A -85,B 0,C 180,E1 -4242.829,E2 -4242.829} C_VEL
LIN {X 0,Y 532.332,Z 287.734,A -85,B 0,C 180,E1 -4243.261,E2 -4243.261} C_VEL
LIN {X 0,Y 532.485,Z 274.075,A -85,B 0,C 180,E1 -4243.549,E2 -4243.549} C_VEL
LIN {X 0,Y 532.737,Z 180.126,A -85,B 0,C 180,E1 -4244.826,E2 -4244.826} C_VEL
LIN {X 0,Y 531.247,Z 171.576,A -85,B 0,C 180,E1 -4244.996,E2 -4244.996} C_VEL
LIN {X 0,Y 531.583,Z 153.414,A -85,B 0,C 180,E1 -4248.28,E2 -4248.28} C_VEL
LIN {X 0,Y 531.592,Z 143.214,A -85,B 0,C 180,E1 -4250.17,E2 -4250.17} C_VEL
LIN {X 0,Y 531.03,Z 139.842,A -85,B 0,C 180,E1 -4250.835,E2 -4250.835} C_VEL
LIN {X 0,Y 530.972,Z 139.843,A -85,B 0,C 180,E1 -4254.225,E2 -4254.225} C_VEL
LIN {X 0,Y 531.002,Z 139.845,A -85,B 0,C 180,E1 -4256.744,E2 -4256.744} C_VEL
LIN {X 0,Y 530.983,Z 139.84,A -85,B 0,C 180,E1 -4259.322,E2 -4259.322} C_VEL
LIN {X 0,Y 530.966,Z 139.843,A -85,B 0,C 180,E1 -4262.1,E2 -4262.1} C_VEL
LIN {X 0,Y 530.97,Z 139.844,A -85,B 0,C 180,E1 -4264.85,E2 -4264.85} C_VEL
LIN {X 0,Y 530.967,Z 139.84,A -85,B 0,C 180,E1 -4267.507,E2 -4267.507} C_VEL
LIN {X 0,Y 530.982,Z 139.846,A -85,B 0,C 180,E1 -4270.433,E2 -4270.433} C_VEL
LIN {X 0,Y 530.966,Z 139.841,A -85,B 0,C 180,E1 -4273.494,E2 -4273.494} C_VEL
LIN {X 0,Y 530.965,Z 139.844,A -85,B 0,C 180,E1 -4276.505,E2 -4276.505} C_VEL
LIN {X 0,Y 530.985,Z 139.841,A -85,B 0,C 180,E1 -4279.567,E2 -4279.567} C_VEL
LIN {X 0,Y 530.968,Z 139.842,A -85,B 0,C 180,E1 -4282.577,E2 -4282.577} C_VEL
LIN {X 0,Y 530.982,Z 139.84,A -85,B 0,C 180,E1 -4285.309,E2 -4285.309} C_VEL
LIN {X 0,Y 530.967,Z 139.846,A -85,B 0,C 180,E1 -4288.032,E2 -4288.032} C_VEL
LIN {X 0,Y 530.989,Z 139.838,A -85,B 0,C 180,E1 -4290.874,E2 -4290.874} C_VEL
LIN {X 0,Y 531.002,Z 139.84,A -85,B 0,C 180,E1 -4293.256,E2 -4293.256} C_VEL
LIN {X 0,Y 530.985,Z 139.841,A -85,B 0,C 180,E1 -4295.96,E2 -4295.96} C_VEL
LIN {X 0,Y 531,Z 139.84,A -85,B 0,C 180,E1 -4299.062,E2 -4299.062} C_VEL
LIN {X 0,Y 531.016,Z 139.834,A -85,B 0,C 180,E1 -4302.278,E2 -4302.278} C_VEL
LIN {X 0,Y 531.019,Z 139.84,A -85,B 0,C 180,E1 -4305.436,E2 -4305.436} C_VEL
LIN {X 0,Y 531.036,Z 139.833,A -85,B 0,C 180,E1 -4308.55,E2 -4308.55} C_VEL
LIN {X 0,Y 531.054,Z 139.831,A -85,B 0,C 180,E1 -4311.629,E2 -4311.629} C_VEL
LIN {X 0,Y 531.12,Z 139.826,A -85,B 0,C 180,E1 -4314.685,E2 -4314.685} C_VEL
LIN {X 0,Y 531.14,Z 139.819,A -85,B 0,C 180,E1 -4317.725,E2 -4317.725} C_VEL
LIN {X 0,Y 531.154,Z 139.826,A -85,B 0,C 180,E1 -4320.758,E2 -4320.758} C_VEL
LIN {X 0,Y 531.103,Z 139.828,A -85,B 0,C 180,E1 -4323.034,E2 -4323.034} C_VEL
LIN {X 0,Y 531.075,Z 139.829,A -85,B 0,C 180,E1 -4326.077,E2 -4326.077} C_VEL
LIN {X 0,Y 531.051,Z 139.836,A -85,B 0,C 180,E1 -4328.371,E2 -4328.371} C_VEL
LIN {X 0,Y 531.051,Z 139.83,A -85,B 0,C 180,E1 -4331.672,E2 -4331.672} C_VEL
LIN {X 0,Y 531.03,Z 139.834,A -85,B 0,C 180,E1 -4334.956,E2 -4334.956} C_VEL
LIN {X 0,Y 530.98,Z 139.841,A -85,B 0,C 180,E1 -4337.724,E2 -4337.724} C_VEL
LIN {X 0,Y 531.024,Z 139.841,A -85,B 0,C 180,E1 -4340.127,E2 -4340.127} C_VEL
LIN {X 0,Y 530.944,Z 139.846,A -85,B 0,C 180,E1 -4342.573,E2 -4342.573} C_VEL
LIN {X 0,Y 530.988,Z 139.838,A -85,B 0,C 180,E1 -4345.059,E2 -4345.059} C_VEL
LIN {X 0,Y 531.007,Z 139.839,A -85,B 0,C 180,E1 -4347.596,E2 -4347.596} C_VEL
LIN {X 0,Y 530.973,Z 139.84,A -85,B 0,C 180,E1 -4350.645,E2 -4350.645} C_VEL
LIN {X 0,Y 530.986,Z 139.847,A -85,B 0,C 180,E1 -4353.773,E2 -4353.773} C_VEL
LIN {X 0,Y 530.95,Z 139.843,A -85,B 0,C 180,E1 -4356.559,E2 -4356.559} C_VEL
LIN {X 0,Y 530.986,Z 139.844,A -85,B 0,C 180,E1 -4359.444,E2 -4359.444} C_VEL
LIN {X 0,Y 530.963,Z 139.841,A -85,B 0,C 180,E1 -4362.458,E2 -4362.458} C_VEL
LIN {X 0,Y 530.967,Z 139.849,A -85,B 0,C 180,E1 -4365.451,E2 -4365.451} C_VEL
LIN {X 0,Y 530.979,Z 139.839,A -85,B 0,C 180,E1 -4368.563,E2 -4368.563} C_VEL
LIN {X 0,Y 530.954,Z 139.847,A -85,B 0,C 180,E1 -4371.529,E2 -4371.529} C_VEL
LIN {X 0,Y 530.954,Z 139.842,A -85,B 0,C 180,E1 -4374.38,E2 -4374.38} C_VEL
LIN {X 0,Y 530.965,Z 139.849,A -85,B 0,C 180,E1 -4377.133,E2 -4377.133} C_VEL
LIN {X 0,Y 530.947,Z 139.845,A -85,B 0,C 180,E1 -4379.802,E2 -4379.802} C_VEL
LIN {X 0,Y 530.964,Z 139.844,A -85,B 0,C 180,E1 -4382.478,E2 -4382.478} C_VEL
LIN {X 0,Y 530.95,Z 139.852,A -85,B 0,C 180,E1 -4384.94,E2 -4384.94} C_VEL
LIN {X 0,Y 530.995,Z 140.03,A -85,B 0,C 180,E1 -4386.331,E2 -4386.331} C_VEL
LIN {X 0,Y 532.201,Z 147.313,A -85,B 0,C 180,E1 -4387.577,E2 -4387.577} C_VEL
LIN {X 0,Y 531.863,Z 163.024,A -85,B 0,C 180,E1 -4390.108,E2 -4390.108} C_VEL
LIN {X 0,Y 531.497,Z 180.547,A -85,B 0,C 180,E1 -4392.89,E2 -4392.89} C_VEL
LIN {X 0,Y 531.27,Z 194.375,A -85,B 0,C 180,E1 -4395.051,E2 -4395.051} C_VEL
LIN {X 0,Y 532.798,Z 204.873,A -85,B 0,C 180,E1 -4395.237,E2 -4395.237} C_VEL
LIN {X 0,Y 532.403,Z 302.3,A -85,B 0,C 180,E1 -4396.571,E2 -4396.571} C_VEL
LIN {X 0,Y 532.215,Z 315.582,A -85,B 0,C 180,E1 -4396.906,E2 -4396.906} C_VEL
LIN {X 0,Y 531.964,Z 328.873,A -85,B 0,C 180,E1 -4397.409,E2 -4397.409} C_VEL
LIN {X 0,Y 531.681,Z 341.219,A -85,B 0,C 180,E1 -4398.057,E2 -4398.057} C_VEL
LIN {X 0,Y 531.439,Z 352.918,A -85,B 0,C 180,E1 -4398.848,E2 -4398.848} C_VEL
LIN {X 0,Y 531.196,Z 363.11,A -85,B 0,C 180,E1 -4399.711,E2 -4399.711} C_VEL
LIN {X 0,Y 530.968,Z 372.279,A -85,B 0,C 180,E1 -4400.669,E2 -4400.669} C_VEL
LIN {X 0,Y 530.775,Z 381.214,A -85,B 0,C 180,E1 -4401.817,E2 -4401.817} C_VEL
LIN {X 0,Y 530.624,Z 388.404,A -85,B 0,C 180,E1 -4402.963,E2 -4402.963} C_VEL
LIN {X 0,Y 530.576,Z 394.952,A -85,B 0,C 180,E1 -4404.299,E2 -4404.299} C_VEL
LIN {X 0,Y 530.45,Z 399.282,A -85,B 0,C 180,E1 -4405.441,E2 -4405.441} C_VEL
LIN {X 0,Y 530.516,Z 401.576,A -85,B 0,C 180,E1 -4406.202,E2 -4406.202} C_VEL
LIN {X 0,Y 530.457,Z 403.433,A -85,B 0,C 180,E1 -4406.962,E2 -4406.962} C_VEL
LIN {X 0,Y 530.411,Z 404.825,A -85,B 0,C 180,E1 -4407.722,E2 -4407.722} C_VEL
LIN {X 0,Y 530.345,Z 406.425,A -85,B 0,C 180,E1 -4409.241,E2 -4409.241} C_VEL
LIN {X 0,Y 530.346,Z 406.641,A -85,B 0,C 180,E1 -4410,E2 -4410} C_VEL
LIN {X 0,Y 530.361,Z 405.82,A -85,B 0,C 180,E1 -4411.519,E2 -4411.519} C_VEL
LIN {X 0,Y 530.411,Z 404.828,A -85,B 0,C 180,E1 -4412.278,E2 -4412.278} C_VEL
LIN {X 0,Y 530.457,Z 403.437,A -85,B 0,C 180,E1 -4413.038,E2 -4413.038} C_VEL
LIN {X 0,Y 530.521,Z 400.508,A -85,B 0,C 180,E1 -4414.178,E2 -4414.178} C_VEL
LIN {X 0,Y 530.522,Z 396.54,A -85,B 0,C 180,E1 -4415.321,E2 -4415.321} C_VEL
LIN {X 0,Y 530.584,Z 390.902,A -85,B 0,C 180,E1 -4416.568,E2 -4416.568} C_VEL
LIN {X 0,Y 530.707,Z 383.771,A -85,B 0,C 180,E1 -4417.801,E2 -4417.801} C_VEL
LIN {X 0,Y 530.898,Z 375.497,A -85,B 0,C 180,E1 -4418.948,E2 -4418.948} C_VEL
LIN {X 0,Y 531.074,Z 367.015,A -85,B 0,C 180,E1 -4419.906,E2 -4419.906} C_VEL
LIN {X 0,Y 531.377,Z 356.535,A -85,B 0,C 180,E1 -4420.864,E2 -4420.864} C_VEL
LIN {X 0,Y 531.648,Z 344.708,A -85,B 0,C 180,E1 -4421.729,E2 -4421.729} C_VEL
LIN {X 0,Y 531.886,Z 332.875,A -85,B 0,C 180,E1 -4422.399,E2 -4422.399} C_VEL
LIN {X 0,Y 532.137,Z 320.533,A -85,B 0,C 180,E1 -4422.926,E2 -4422.926} C_VEL
LIN {X 0,Y 532.336,Z 307.87,A -85,B 0,C 180,E1 -4423.31,E2 -4423.31} C_VEL
LIN {X 0,Y 532.494,Z 294.657,A -85,B 0,C 180,E1 -4423.549,E2 -4423.549} C_VEL
LIN {X 0,Y 532.629,Z 203.131,A -85,B 0,C 180,E1 -4424.791,E2 -4424.791} C_VEL
LIN {X 0,Y 531.269,Z 194.176,A -85,B 0,C 180,E1 -4424.968,E2 -4424.968} C_VEL
LIN {X 0,Y 531.635,Z 174.235,A -85,B 0,C 180,E1 -4428.108,E2 -4428.108} C_VEL
LIN {X 0,Y 532.061,Z 155.511,A -85,B 0,C 180,E1 -4431.097,E2 -4431.097} C_VEL
LIN {X 0,Y 532.212,Z 146.738,A -85,B 0,C 180,E1 -4432.517,E2 -4432.517} C_VEL
LIN {X 0,Y 530.994,Z 139.844,A -85,B 0,C 180,E1 -4433.715,E2 -4433.715} C_VEL
LIN {X 0,Y 530.967,Z 139.846,A -85,B 0,C 180,E1 -4436.746,E2 -4436.746} C_VEL
LIN {X 0,Y 530.961,Z 139.845,A -85,B 0,C 180,E1 -4439.324,E2 -4439.324} C_VEL
LIN {X 0,Y 530.957,Z 139.842,A -85,B 0,C 180,E1 -4442.098,E2 -4442.098} C_VEL
LIN {X 0,Y 530.968,Z 139.849,A -85,B 0,C 180,E1 -4444.85,E2 -4444.85} C_VEL
LIN {X 0,Y 530.965,Z 139.841,A -85,B 0,C 180,E1 -4447.508,E2 -4447.508} C_VEL
LIN {X 0,Y 530.961,Z 139.846,A -85,B 0,C 180,E1 -4450.435,E2 -4450.435} C_VEL
LIN {X 0,Y 530.933,Z 139.846,A -85,B 0,C 180,E1 -4453.278,E2 -4453.278} C_VEL
LIN {X 0,Y 530.975,Z 139.839,A -85,B 0,C 180,E1 -4455.622,E2 -4455.622} C_VEL
LIN {X 0,Y 530.986,Z 139.846,A -85,B 0,C 180,E1 -4458.563,E2 -4458.563} C_VEL
LIN {X 0,Y 530.955,Z 139.842,A -85,B 0,C 180,E1 -4461.529,E2 -4461.529} C_VEL
LIN {X 0,Y 530.95,Z 139.85,A -85,B 0,C 180,E1 -4464.379,E2 -4464.379} C_VEL
LIN {X 0,Y 530.967,Z 139.84,A -85,B 0,C 180,E1 -4467.133,E2 -4467.133} C_VEL
LIN {X 0,Y 530.958,Z 139.846,A -85,B 0,C 180,E1 -4469.802,E2 -4469.802} C_VEL
LIN {X 0,Y 530.974,Z 139.843,A -85,B 0,C 180,E1 -4472.475,E2 -4472.475} C_VEL
LIN {X 0,Y 530.987,Z 139.838,A -85,B 0,C 180,E1 -4474.941,E2 -4474.941} C_VEL
LIN {X 0,Y 530.971,Z 139.844,A -85,B 0,C 180,E1 -4478.247,E2 -4478.247} C_VEL
LIN {X 0,Y 530.991,Z 139.838,A -85,B 0,C 180,E1 -4480.677,E2 -4480.677} C_VEL
LIN {X 0,Y 530.969,Z 139.841,A -85,B 0,C 180,E1 -4483.07,E2 -4483.07} C_VEL
LIN {X 0,Y 531.019,Z 139.84,A -85,B 0,C 180,E1 -4485.436,E2 -4485.436} C_VEL
LIN {X 0,Y 531.037,Z 139.832,A -85,B 0,C 180,E1 -4488.55,E2 -4488.55} C_VEL
LIN {X 0,Y 531.052,Z 139.837,A -85,B 0,C 180,E1 -4491.629,E2 -4491.629} C_VEL
LIN {X 0,Y 531.121,Z 139.822,A -85,B 0,C 180,E1 -4494.685,E2 -4494.685} C_VEL
LIN {X 0,Y 531.142,Z 139.822,A -85,B 0,C 180,E1 -4497.725,E2 -4497.725} C_VEL
LIN {X 0,Y 531.15,Z 139.82,A -85,B 0,C 180,E1 -4500.758,E2 -4500.758} C_VEL
LIN {X 0,Y 531.104,Z 139.831,A -85,B 0,C 180,E1 -4503.034,E2 -4503.034} C_VEL
LIN {X 0,Y 531.074,Z 139.827,A -85,B 0,C 180,E1 -4506.077,E2 -4506.077} C_VEL
LIN {X 0,Y 531.053,Z 139.831,A -85,B 0,C 180,E1 -4508.371,E2 -4508.371} C_VEL
LIN {X 0,Y 531.052,Z 139.83,A -85,B 0,C 180,E1 -4511.672,E2 -4511.672} C_VEL
LIN {X 0,Y 531.031,Z 139.839,A -85,B 0,C 180,E1 -4514.956,E2 -4514.956} C_VEL
LIN {X 0,Y 531.017,Z 139.834,A -85,B 0,C 180,E1 -4517.722,E2 -4517.722} C_VEL
LIN {X 0,Y 531,Z 139.84,A -85,B 0,C 180,E1 -4520.938,E2 -4520.938} C_VEL
LIN {X 0,Y 530.972,Z 139.845,A -85,B 0,C 180,E1 -4524.225,E2 -4524.225} C_VEL
LIN {X 0,Y 531.002,Z 139.84,A -85,B 0,C 180,E1 -4526.744,E2 -4526.744} C_VEL
LIN {X 0,Y 530.982,Z 139.838,A -85,B 0,C 180,E1 -4529.323,E2 -4529.323} C_VEL
LIN {X 0,Y 530.966,Z 139.847,A -85,B 0,C 180,E1 -4532.101,E2 -4532.101} C_VEL
LIN {X 0,Y 530.971,Z 139.841,A -85,B 0,C 180,E1 -4534.851,E2 -4534.851} C_VEL
LIN {X 0,Y 530.967,Z 139.842,A -85,B 0,C 180,E1 -4537.508,E2 -4537.508} C_VEL
LIN {X 0,Y 530.985,Z 139.841,A -85,B 0,C 180,E1 -4540.433,E2 -4540.433} C_VEL
LIN {X 0,Y 530.966,Z 139.843,A -85,B 0,C 180,E1 -4543.495,E2 -4543.495} C_VEL
LIN {X 0,Y 530.964,Z 139.843,A -85,B 0,C 180,E1 -4543.552,E2 -4543.552} C_VEL
LIN {X 0,Y 530.291,Z 139.93,A -85,B 0,C 180,E1 -4544.185,E2 -4544.185} C_VEL
LIN {X 0,Y 527.444,Z 140.28,A -85,B 0,C 180,E1 -4545.214,E2 -4545.214} C_VEL
LIN {X 0,Y 525.041,Z 140.585,A -85,B 0,C 180,E1 -4546.042,E2 -4546.042} C_VEL
LIN {X 0,Y 524.007,Z 140.708,A -85,B 0,C 180,E1 -4546.682,E2 -4546.682} C_VEL
LIN {X 0,Y 523.921,Z 140.718,A -85,B 0,C 180,E1 -4546.898,E2 -4546.898} C_VEL
LIN {X 0,Y 523.95,Z 140.721,A -85,B 0,C 180,E1 -4549.921,E2 -4549.921} C_VEL
LIN {X 0,Y 523.909,Z 140.72,A -85,B 0,C 180,E1 -4552.868,E2 -4552.868} C_VEL
LIN {X 0,Y 523.922,Z 140.725,A -85,B 0,C 180,E1 -4555.709,E2 -4555.709} C_VEL
LIN {X 0,Y 523.921,Z 140.718,A -85,B 0,C 180,E1 -4558.456,E2 -4558.456} C_VEL
LIN {X 0,Y 523.937,Z 140.721,A -85,B 0,C 180,E1 -4561.125,E2 -4561.125} C_VEL
LIN {X 0,Y 523.987,Z 140.712,A -85,B 0,C 180,E1 -4563.981,E2 -4563.981} C_VEL
LIN {X 0,Y 523.927,Z 140.719,A -85,B 0,C 180,E1 -4566.27,E2 -4566.27} C_VEL
LIN {X 0,Y 523.989,Z 140.807,A -85,B 0,C 180,E1 -4569.154,E2 -4569.154} C_VEL
LIN {X 0,Y 524.708,Z 145.542,A -85,B 0,C 180,E1 -4570.081,E2 -4570.081} C_VEL
LIN {X 0,Y 524.461,Z 159.398,A -85,B 0,C 180,E1 -4572.657,E2 -4572.657} C_VEL
LIN {X 0,Y 524.257,Z 171.728,A -85,B 0,C 180,E1 -4574.898,E2 -4574.898} C_VEL
LIN {X 0,Y 526.008,Z 182.257,A -85,B 0,C 180,E1 -4575.098,E2 -4575.098} C_VEL
LIN {X 0,Y 525.548,Z 278.995,A -85,B 0,C 180,E1 -4576.441,E2 -4576.441} C_VEL
LIN {X 0,Y 525.368,Z 292.179,A -85,B 0,C 180,E1 -4576.781,E2 -4576.781} C_VEL
LIN {X 0,Y 525.131,Z 304.281,A -85,B 0,C 180,E1 -4577.243,E2 -4577.243} C_VEL
LIN {X 0,Y 524.924,Z 316.543,A -85,B 0,C 180,E1 -4577.879,E2 -4577.879} C_VEL
LIN {X 0,Y 524.647,Z 327.377,A -85,B 0,C 180,E1 -4578.604,E2 -4578.604} C_VEL
LIN {X 0,Y 524.34,Z 337.861,A -85,B 0,C 180,E1 -4579.477,E2 -4579.477} C_VEL
LIN {X 0,Y 524.1,Z 346.426,A -85,B 0,C 180,E1 -4580.35,E2 -4580.35} C_VEL
LIN {X 0,Y 523.897,Z 354.314,A -85,B 0,C 180,E1 -4581.32,E2 -4581.32} C_VEL
LIN {X 0,Y 523.678,Z 362.03,A -85,B 0,C 180,E1 -4582.481,E2 -4582.481} C_VEL
LIN {X 0,Y 523.593,Z 369.104,A -85,B 0,C 180,E1 -4583.836,E2 -4583.836} C_VEL
LIN {X 0,Y 523.387,Z 373.823,A -85,B 0,C 180,E1 -4584.993,E2 -4584.993} C_VEL
LIN {X 0,Y 523.445,Z 377.433,A -85,B 0,C 180,E1 -4586.151,E2 -4586.151} C_VEL
LIN {X 0,Y 523.417,Z 379.301,A -85,B 0,C 180,E1 -4586.921,E2 -4586.921} C_VEL
LIN {X 0,Y 523.338,Z 380.712,A -85,B 0,C 180,E1 -4587.691,E2 -4587.691} C_VEL
LIN {X 0,Y 523.253,Z 382.333,A -85,B 0,C 180,E1 -4589.23,E2 -4589.23} C_VEL
LIN {X 0,Y 523.251,Z 382.571,A -85,B 0,C 180,E1 -4590,E2 -4590} C_VEL
LIN {X 0,Y 523.253,Z 382.388,A -85,B 0,C 180,E1 -4590.77,E2 -4590.77} C_VEL
LIN {X 0,Y 523.338,Z 380.84,A -85,B 0,C 180,E1 -4592.309,E2 -4592.309} C_VEL
LIN {X 0,Y 523.417,Z 379.484,A -85,B 0,C 180,E1 -4593.079,E2 -4593.079} C_VEL
LIN {X 0,Y 523.446,Z 376.62,A -85,B 0,C 180,E1 -4594.235,E2 -4594.235} C_VEL
LIN {X 0,Y 523.465,Z 372.737,A -85,B 0,C 180,E1 -4595.393,E2 -4595.393} C_VEL
LIN {X 0,Y 523.555,Z 367.445,A -85,B 0,C 180,E1 -4596.611,E2 -4596.611} C_VEL
LIN {X 0,Y 523.739,Z 360.195,A -85,B 0,C 180,E1 -4597.906,E2 -4597.906} C_VEL
LIN {X 0,Y 523.924,Z 352.042,A -85,B 0,C 180,E1 -4599.068,E2 -4599.068} C_VEL
LIN {X 0,Y 524.165,Z 343.696,A -85,B 0,C 180,E1 -4600.038,E2 -4600.038} C_VEL
LIN {X 0,Y 524.47,Z 333.394,A -85,B 0,C 180,E1 -4601.008,E2 -4601.008} C_VEL
LIN {X 0,Y 524.75,Z 322.858,A -85,B 0,C 180,E1 -4601.808,E2 -4601.808} C_VEL
LIN {X 0,Y 525.013,Z 312.027,A -85,B 0,C 180,E1 -4602.466,E2 -4602.466} C_VEL
LIN {X 0,Y 525.222,Z 300.717,A -85,B 0,C 180,E1 -4603.001,E2 -4603.001} C_VEL
LIN {X 0,Y 525.439,Z 287.873,A -85,B 0,C 180,E1 -4603.438,E2 -4603.438} C_VEL
LIN {X 0,Y 525.598,Z 274.199,A -85,B 0,C 180,E1 -4603.73,E2 -4603.73} C_VEL
LIN {X 0,Y 525.946,Z 181.356,A -85,B 0,C 180,E1 -4605.006,E2 -4605.006} C_VEL
LIN {X 0,Y 524.241,Z 171.712,A -85,B 0,C 180,E1 -4605.196,E2 -4605.196} C_VEL
LIN {X 0,Y 524.589,Z 154.412,A -85,B 0,C 180,E1 -4608.351,E2 -4608.351} C_VEL
LIN {X 0,Y 524.545,Z 144.036,A -85,B 0,C 180,E1 -4610.301,E2 -4610.301} C_VEL
LIN {X 0,Y 524.002,Z 140.717,A -85,B 0,C 180,E1 -4610.973,E2 -4610.973} C_VEL
LIN {X 0,Y 523.955,Z 140.717,A -85,B 0,C 180,E1 -4614.201,E2 -4614.201} C_VEL
LIN {X 0,Y 523.951,Z 140.718,A -85,B 0,C 180,E1 -4617.133,E2 -4617.133} C_VEL
LIN {X 0,Y 523.94,Z 140.716,A -85,B 0,C 180,E1 -4619.756,E2 -4619.756} C_VEL
LIN {X 0,Y 523.935,Z 140.724,A -85,B 0,C 180,E1 -4622.449,E2 -4622.449} C_VEL
LIN {X 0,Y 523.921,Z 140.719,A -85,B 0,C 180,E1 -4625.226,E2 -4625.226} C_VEL
LIN {X 0,Y 523.917,Z 140.723,A -85,B 0,C 180,E1 -4628.101,E2 -4628.101} C_VEL
LIN {X 0,Y 523.94,Z 140.716,A -85,B 0,C 180,E1 -4631.092,E2 -4631.092} C_VEL
LIN {X 0,Y 523.942,Z 140.725,A -85,B 0,C 180,E1 -4634.227,E2 -4634.227} C_VEL
LIN {X 0,Y 523.922,Z 140.719,A -85,B 0,C 180,E1 -4636.833,E2 -4636.833} C_VEL
LIN {X 0,Y 523.942,Z 140.716,A -85,B 0,C 180,E1 -4638.908,E2 -4638.908} C_VEL
LIN {X 0,Y 523.917,Z 140.727,A -85,B 0,C 180,E1 -4641.898,E2 -4641.898} C_VEL
LIN {X 0,Y 523.924,Z 140.718,A -85,B 0,C 180,E1 -4644.911,E2 -4644.911} C_VEL
LIN {X 0,Y 523.935,Z 140.724,A -85,B 0,C 180,E1 -4647.679,E2 -4647.679} C_VEL
LIN {X 0,Y 523.954,Z 140.714,A -85,B 0,C 180,E1 -4650.676,E2 -4650.676} C_VEL
LIN {X 0,Y 523.974,Z 140.719,A -85,B 0,C 180,E1 -4653.728,E2 -4653.728} C_VEL
LIN {X 0,Y 523.926,Z 140.718,A -85,B 0,C 180,E1 -4656.27,E2 -4656.27} C_VEL
LIN {X 0,Y 523.946,Z 140.716,A -85,B 0,C 180,E1 -4658.767,E2 -4658.767} C_VEL
LIN {X 0,Y 523.951,Z 140.721,A -85,B 0,C 180,E1 -4661.221,E2 -4661.221} C_VEL
LIN {X 0,Y 523.937,Z 140.72,A -85,B 0,C 180,E1 -4663.639,E2 -4663.639} C_VEL
LIN {X 0,Y 523.939,Z 140.716,A -85,B 0,C 180,E1 -4666.028,E2 -4666.028} C_VEL
LIN {X 0,Y 524.012,Z 140.707,A -85,B 0,C 180,E1 -4668.394,E2 -4668.394} C_VEL
LIN {X 0,Y 524.003,Z 140.711,A -85,B 0,C 180,E1 -4671.516,E2 -4671.516} C_VEL
LIN {X 0,Y 524.081,Z 140.702,A -85,B 0,C 180,E1 -4674.614,E2 -4674.614} C_VEL
LIN {X 0,Y 524.112,Z 140.695,A -85,B 0,C 180,E1 -4677.694,E2 -4677.694} C_VEL
LIN {X 0,Y 524.123,Z 140.702,A -85,B 0,C 180,E1 -4680.768,E2 -4680.768} C_VEL
LIN {X 0,Y 524.069,Z 140.704,A -85,B 0,C 180,E1 -4683.075,E2 -4683.075} C_VEL
LIN {X 0,Y 524.037,Z 140.706,A -85,B 0,C 180,E1 -4686.159,E2 -4686.159} C_VEL
LIN {X 0,Y 524,Z 140.716,A -85,B 0,C 180,E1 -4688.484,E2 -4688.484} C_VEL
LIN {X 0,Y 524.002,Z 140.709,A -85,B 0,C 180,E1 -4691.739,E2 -4691.739} C_VEL
LIN {X 0,Y 523.992,Z 140.71,A -85,B 0,C 180,E1 -4695.052,E2 -4695.052} C_VEL
LIN {X 0,Y 523.946,Z 140.72,A -85,B 0,C 180,E1 -4697.97,E2 -4697.97} C_VEL
LIN {X 0,Y 523.971,Z 140.718,A -85,B 0,C 180,E1 -4700.41,E2 -4700.41} C_VEL
LIN {X 0,Y 523.91,Z 140.72,A -85,B 0,C 180,E1 -4702.894,E2 -4702.894} C_VEL
LIN {X 0,Y 523.981,Z 140.72,A -85,B 0,C 180,E1 -4706.019,E2 -4706.019} C_VEL
LIN {X 0,Y 523.928,Z 140.717,A -85,B 0,C 180,E1 -4708.875,E2 -4708.875} C_VEL
LIN {X 0,Y 523.92,Z 140.723,A -85,B 0,C 180,E1 -4711.544,E2 -4711.544} C_VEL
LIN {X 0,Y 523.931,Z 140.719,A -85,B 0,C 180,E1 -4714.29,E2 -4714.29} C_VEL
LIN {X 0,Y 523.904,Z 140.722,A -85,B 0,C 180,E1 -4717.133,E2 -4717.133} C_VEL
LIN {X 0,Y 523.937,Z 140.718,A -85,B 0,C 180,E1 -4720.13,E2 -4720.13} C_VEL
LIN {X 0,Y 523.921,Z 140.718,A -85,B 0,C 180,E1 -4722.457,E2 -4722.457} C_VEL
LIN {X 0,Y 523.938,Z 140.723,A -85,B 0,C 180,E1 -4725.311,E2 -4725.311} C_VEL
LIN {X 0,Y 523.939,Z 140.717,A -85,B 0,C 180,E1 -4728.692,E2 -4728.692} C_VEL
LIN {X 0,Y 523.913,Z 140.72,A -85,B 0,C 180,E1 -4731.898,E2 -4731.898} C_VEL
LIN {X 0,Y 523.923,Z 140.723,A -85,B 0,C 180,E1 -4734.912,E2 -4734.912} C_VEL
LIN {X 0,Y 523.931,Z 140.718,A -85,B 0,C 180,E1 -4737.681,E2 -4737.681} C_VEL
LIN {X 0,Y 523.936,Z 140.723,A -85,B 0,C 180,E1 -4740.681,E2 -4740.681} C_VEL
LIN {X 0,Y 523.909,Z 140.723,A -85,B 0,C 180,E1 -4743.725,E2 -4743.725} C_VEL
LIN {X 0,Y 523.96,Z 140.91,A -85,B 0,C 180,E1 -4746.167,E2 -4746.167} C_VEL
LIN {X 0,Y 525.231,Z 148.05,A -85,B 0,C 180,E1 -4747.41,E2 -4747.41} C_VEL
LIN {X 0,Y 524.898,Z 164.126,A -85,B 0,C 180,E1 -4750.036,E2 -4750.036} C_VEL
LIN {X 0,Y 524.474,Z 181.64,A -85,B 0,C 180,E1 -4752.854,E2 -4752.854} C_VEL
LIN {X 0,Y 524.25,Z 194.142,A -85,B 0,C 180,E1 -4754.845,E2 -4754.845} C_VEL
LIN {X 0,Y 525.926,Z 205.496,A -85,B 0,C 180,E1 -4755.051,E2 -4755.051} C_VEL
LIN {X 0,Y 525.515,Z 302.139,A -85,B 0,C 180,E1 -4756.391,E2 -4756.391} C_VEL
LIN {X 0,Y 525.293,Z 315.42,A -85,B 0,C 180,E1 -4756.73,E2 -4756.73} C_VEL
LIN {X 0,Y 525.034,Z 328.71,A -85,B 0,C 180,E1 -4757.24,E2 -4757.24} C_VEL
LIN {X 0,Y 524.715,Z 341.027,A -85,B 0,C 180,E1 -4757.894,E2 -4757.894} C_VEL
LIN {X 0,Y 524.461,Z 352.756,A -85,B 0,C 180,E1 -4758.698,E2 -4758.698} C_VEL
LIN {X 0,Y 524.163,Z 362.946,A -85,B 0,C 180,E1 -4759.572,E2 -4759.572} C_VEL
LIN {X 0,Y 523.944,Z 372.117,A -85,B 0,C 180,E1 -4760.543,E2 -4760.543} C_VEL
LIN {X 0,Y 523.721,Z 381.051,A -85,B 0,C 180,E1 -4761.706,E2 -4761.706} C_VEL
LIN {X 0,Y 523.569,Z 388.242,A -85,B 0,C 180,E1 -4762.868,E2 -4762.868} C_VEL
LIN {X 0,Y 523.476,Z 393.094,A -85,B 0,C 180,E1 -4763.834,E2 -4763.834} C_VEL
LIN {X 0,Y 523.383,Z 397.809,A -85,B 0,C 180,E1 -4764.993,E2 -4764.993} C_VEL
LIN {X 0,Y 523.443,Z 401.414,A -85,B 0,C 180,E1 -4766.151,E2 -4766.151} C_VEL
LIN {X 0,Y 523.367,Z 403.271,A -85,B 0,C 180,E1 -4766.921,E2 -4766.921} C_VEL
LIN {X 0,Y 523.335,Z 404.664,A -85,B 0,C 180,E1 -4767.691,E2 -4767.691} C_VEL
LIN {X 0,Y 523.251,Z 406.263,A -85,B 0,C 180,E1 -4769.23,E2 -4769.23} C_VEL
LIN {X 0,Y 523.25,Z 406.479,A -85,B 0,C 180,E1 -4770,E2 -4770} C_VEL
LIN {X 0,Y 523.275,Z 405.658,A -85,B 0,C 180,E1 -4771.539,E2 -4771.539} C_VEL
LIN {X 0,Y 523.335,Z 404.667,A -85,B 0,C 180,E1 -4772.309,E2 -4772.309} C_VEL
LIN {X 0,Y 523.367,Z 403.274,A -85,B 0,C 180,E1 -4773.079,E2 -4773.079} C_VEL
LIN {X 0,Y 523.423,Z 400.345,A -85,B 0,C 180,E1 -4774.235,E2 -4774.235} C_VEL
LIN {X 0,Y 523.456,Z 396.378,A -85,B 0,C 180,E1 -4775.393,E2 -4775.393} C_VEL
LIN {X 0,Y 523.504,Z 391.223,A -85,B 0,C 180,E1 -4776.563,E2 -4776.563} C_VEL
LIN {X 0,Y 523.63,Z 384.844,A -85,B 0,C 180,E1 -4777.713,E2 -4777.713} C_VEL
LIN {X 0,Y 523.803,Z 376.824,A -85,B 0,C 180,E1 -4778.876,E2 -4778.876} C_VEL
LIN {X 0,Y 524.016,Z 368.651,A -85,B 0,C 180,E1 -4779.846,E2 -4779.846} C_VEL
LIN {X 0,Y 524.329,Z 358.685,A -85,B 0,C 180,E1 -4780.816,E2 -4780.816} C_VEL
LIN {X 0,Y 524.6,Z 347.504,A -85,B 0,C 180,E1 -4781.686,E2 -4781.686} C_VEL
LIN {X 0,Y 524.843,Z 336.404,A -85,B 0,C 180,E1 -4782.372,E2 -4782.372} C_VEL
LIN {X 0,Y 525.132,Z 324.184,A -85,B 0,C 180,E1 -4782.954,E2 -4782.954} C_VEL
LIN {X 0,Y 525.366,Z 311.369,A -85,B 0,C 180,E1 -4783.391,E2 -4783.391} C_VEL
LIN {X 0,Y 525.568,Z 297.786,A -85,B 0,C 180,E1 -4783.681,E2 -4783.681} C_VEL
LIN {X 0,Y 525.838,Z 204.231,A -85,B 0,C 180,E1 -4784.969,E2 -4784.969} C_VEL
LIN {X 0,Y 524.228,Z 194.077,A -85,B 0,C 180,E1 -4785.164,E2 -4785.164} C_VEL
LIN {X 0,Y 524.637,Z 175.512,A -85,B 0,C 180,E1 -4788.127,E2 -4788.127} C_VEL
LIN {X 0,Y 525.119,Z 156.612,A -85,B 0,C 180,E1 -4791.184,E2 -4791.184} C_VEL
LIN {X 0,Y 525.256,Z 148.002,A -85,B 0,C 180,E1 -4792.597,E2 -4792.597} C_VEL
LIN {X 0,Y 523.948,Z 140.721,A -85,B 0,C 180,E1 -4793.868,E2 -4793.868} C_VEL
LIN {X 0,Y 523.909,Z 140.727,A -85,B 0,C 180,E1 -4797.135,E2 -4797.135} C_VEL
